			(* Case 60 - AspirazioneDX *)
			60: 
				IF AspirazioneSX1^.Status.CommandDone AND AspirazioneDX1^.Status.CommandDone AND
					AspirazioneSX2^.Status.CommandDone AND AspirazioneDX2^.Status.CommandDone THEN
					AspirazioneDX1^.Command^.Aspirazione_ON 	:= FALSE;
					AspirazioneDX1^.Command^.Aspirazione_OFF	:= FALSE;
					AspirazioneSX1^.Command^.Aspirazione_ON 	:= FALSE;
					AspirazioneSX1^.Command^.Aspirazione_OFF	:= FALSE;
					AspirazioneDX2^.Command^.Aspirazione_ON 	:= FALSE;
					AspirazioneDX2^.Command^.Aspirazione_OFF	:= FALSE;
					AspirazioneSX2^.Command^.Aspirazione_ON 	:= FALSE;
					AspirazioneSX2^.Command^.Aspirazione_OFF	:= FALSE;
					TFCommandCase(ADR(CmdExe),100,CommandCase_JMP);
				ELSIF AspirazioneSX1^.Status.ErrorID <> ErrNULL THEN
					TFClearAllCmdModulePinzaCompleta(AspirazioneDX1,AspirazioneSX1,AspirazioneDX2,AspirazioneSX2,CilindroApertura,CilindroSbloccoRotazione,CilindroSbloccoBascolante,AspirazioneFaldaDX,AspirazioneFaldaSX);
					TFError(ErrCYLINDER,AspirazioneSX1^.Status.ErrorID,ADR(CmdExe),ADR(State),ADR(Error),ADR(ErrorLog));
				ELSIF AspirazioneDX1^.Status.ErrorID <> ErrNULL THEN
					TFClearAllCmdModulePinzaCompleta(AspirazioneDX1,AspirazioneSX1,AspirazioneDX2,AspirazioneSX2,CilindroApertura,CilindroSbloccoRotazione,CilindroSbloccoBascolante,AspirazioneFaldaDX,AspirazioneFaldaSX);
					TFError(ErrCYLINDER,AspirazioneDX1^.Status.ErrorID,ADR(CmdExe),ADR(State),ADR(Error),ADR(ErrorLog));
				END_IF

			(* Case 70 - CilindroTasteggio *)
			70: 
				//IF CilindroTasteggio^.Status.CommandDone THEN
				//	CilindroTasteggio^.Command.Activation 		:= FALSE;
				//	CilindroTasteggio^.Command.Deactivation 	:= FALSE;
					TFCommandCase(ADR(CmdExe),100,CommandCase_JMP);
				//END_IF								
				
			(* Case 100 - End *)
			100:(* Clear All Output Here *)
				TFStateUpdate(ADR(State),StateMAN_END);
				TFCommandExeClear(ADR(CmdExe));

			ELSE
				TFError(ErrNOCMDCASE,ErrNULL,ADR(CmdExe),ADR(State),ADR(Error),ADR(ErrorLog));
		END_CASE;

		IF TFTimerDone(ADR(Timeout)) THEN
			TFClearAllCmdModulePinzaCompleta(AspirazioneDX1,AspirazioneSX1,AspirazioneDX2,AspirazioneSX2,CilindroApertura,CilindroSbloccoRotazione,CilindroSbloccoBascolante,AspirazioneFaldaDX,AspirazioneFaldaSX);
			TFError(ErrCMDTIMEOUT,ErrNULL,ADR(CmdExe),ADR(State),ADR(Error),ADR(ErrorLog));
		END_IF
	

	(* ******************************************************************************************************** *)
	(* PRELOAD - Presa del pezzo *)
	(* ******************************************************************************************************** *)
	CmdPRELOAD:
		CASE CmdExe.CmdCase OF
			
			(* Case 0 - Init Command*)
			0: 	TFStateUpdate(ADR(State),StatePRELOAD_RUN);
				TFTimerSet(ADR(Timeout),30000+200,TRUE);
				TFTimerSet(ADR(Timer),30000,TRUE);
				PrelievoSuCavallina := FALSE;
				StatoPinza.ElementoPrelevato := FALSE;
				IF TFCommandParRead(CmdExe.Cmd.Parameter,ADR(ParametersArray),2) THEN
					PrelievoSuCavallina	:= STRING_TO_BOOL(ParametersArray.Parameters[0]);
					AspiraSoloFalde		:= STRING_TO_BOOL(ParametersArray.Parameters[1]);
					TFCommandCase(ADR(CmdExe),10,CommandCase_JMP);
				ELSE
					TFError(ErrCMDPARNUM,ErrNULL,ADR(CmdExe),ADR(State),ADR(Error),ADR(ErrorLog));
					RETURN;
				END_IF;
				
			(* Case 10 - CilindroApertura *)
			10: 
				IF (ElementoInPrelievo.Typology = QUADROTTA OR ElementoInPrelievo.XDim >= 2700) AND AbilitaAperturaAutomaticaPinza THEN //sE HO LE CONDIZIONI APRO LA PINZA
					CilindroApertura^.Command.Activation 	:= TRUE;
					CilindroApertura^.Command.Deactivation 	:= FALSE;
	
					IF CilindroApertura^.Status.Active THEN
						CilindroApertura^.Command.Activation 	:= FALSE;
						CilindroApertura^.Command.Deactivation 	:= FALSE;
						TFCommandCase(ADR(CmdExe),20,CommandCase_JMP);
					ELSIF CilindroApertura^.Status.ErrorID <> ErrNULL THEN
						TFClearAllCmdModulePinzaCompleta(AspirazioneDX1,AspirazioneSX1,AspirazioneDX2,AspirazioneSX2,CilindroApertura,CilindroSbloccoRotazione,CilindroSbloccoBascolante,AspirazioneFaldaDX,AspirazioneFaldaSX);
						TFError(ErrCYLINDER,CilindroApertura^.Status.ErrorID,ADR(CmdExe),ADR(State),ADR(Error),ADR(ErrorLog));
					END_IF
				ELSE

					CilindroApertura^.Command.Activation 	:= FALSE;
					CilindroApertura^.Command.Deactivation 	:= TRUE;
	
					IF CilindroApertura^.Status.Inactive THEN
						CilindroApertura^.Command.Activation 	:= FALSE;
						CilindroApertura^.Command.Deactivation 	:= FALSE;
						TFCommandCase(ADR(CmdExe),20,CommandCase_JMP);
					ELSIF CilindroApertura^.Status.ErrorID <> ErrNULL THEN
						TFClearAllCmdModulePinzaCompleta(AspirazioneDX1,AspirazioneSX1,AspirazioneDX2,AspirazioneSX2,CilindroApertura,CilindroSbloccoRotazione,CilindroSbloccoBascolante,AspirazioneFaldaDX,AspirazioneFaldaSX);
						TFError(ErrCYLINDER,CilindroApertura^.Status.ErrorID,ADR(CmdExe),ADR(State),ADR(Error),ADR(ErrorLog));
					END_IF
					
				END_IF

			(* Case 20 - CilindroSbloccoRotazione *)
			20: 
				IF PrelievoSuCavallina THEN
					CilindroSbloccoRotazione^.Command.Activation 	:= AbilitazioneSbloccoRotazione;
					CilindroSbloccoRotazione^.Command.Deactivation 	:= FALSE;
	
					//CilindroTasteggio^.Command.Activation 		:= AbilitazioneCilindriTastatori;
					//CilindroTasteggio^.Command.Deactivation 	:= FALSE;
					
					IF (CilindroSbloccoRotazione^.Status.Active OR NOT AbilitazioneSbloccoRotazione) THEN
						CilindroSbloccoRotazione^.Command.Activation 	:= FALSE;
						CilindroSbloccoRotazione^.Command.Deactivation 	:= FALSE;
						//CilindroTasteggio^.Command.Activation 		:= FALSE;
						//CilindroTasteggio^.Command.Deactivation 	:= FALSE;
						TFCommandCase(ADR(CmdExe),30,CommandCase_JMP);
					ELSIF CilindroSbloccoRotazione^.Status.ErrorID <> ErrNULL AND AbilitazioneSbloccoRotazione THEN
						TFClearAllCmdModulePinzaCompleta(AspirazioneDX1,AspirazioneSX1,AspirazioneDX2,AspirazioneSX2,CilindroApertura,CilindroSbloccoRotazione,CilindroSbloccoBascolante,AspirazioneFaldaDX,AspirazioneFaldaSX);
						TFError(ErrCYLINDER,CilindroSbloccoRotazione^.Status.ErrorID,ADR(CmdExe),ADR(State),ADR(Error),ADR(ErrorLog));
					//ELSIF CilindroTasteggio^.Status.ErrorID <> ErrNULL THEN
					//	TFClearAllCmdModulePinzaCompleta(AspirazioneDX,AspirazioneSX,CilindroApertura,CilindroSbloccoRotazione,AspirazioneFaldaDX,AspirazioneFaldaSX);
					//	TFError(ErrCYLINDER,CilindroTasteggio^.Status.ErrorID,ADR(CmdExe),ADR(State),ADR(Error),ADR(ErrorLog));
					END_IF

				ELSE
					TFCommandCase(ADR(CmdExe),30,CommandCase_JMP);
				END_IF

			(* Case 30 - AspirazioneFaldaDX *)
			30: 

				IF NOT PrelievoSuCavallina AND AspiraSoloFalde THEN
					AspirazioneFaldaDX^.Command.Activation 	:= TRUE;
					AspirazioneFaldaDX^.Command.Deactivation 	:= FALSE;
					AspirazioneFaldaSX^.Command.Activation 	:= TRUE;
					AspirazioneFaldaSX^.Command.Deactivation 	:= FALSE;
					
					IF AspirazioneFaldaDX^.Status.Active AND AspirazioneFaldaSX^.Status.Active THEN
						AspirazioneFaldaDX^.Command.Activation 	:= FALSE;
						AspirazioneFaldaDX^.Command.Deactivation 	:= FALSE;
						AspirazioneFaldaSX^.Command.Activation 	:= FALSE;
						AspirazioneFaldaSX^.Command.Deactivation 	:= FALSE;
						TFCommandCase(ADR(CmdExe),40,CommandCase_JMP);
					ELSIF AspirazioneFaldaDX^.Status.ErrorID <> ErrNULL THEN
						TFClearAllCmdModulePinzaCompleta(AspirazioneDX1,AspirazioneSX1,AspirazioneDX2,AspirazioneSX2,CilindroApertura,CilindroSbloccoRotazione,CilindroSbloccoBascolante,AspirazioneFaldaDX,AspirazioneFaldaSX);
						TFError(ErrCYLINDER,AspirazioneFaldaDX^.Status.ErrorID,ADR(CmdExe),ADR(State),ADR(Error),ADR(ErrorLog));
					ELSIF AspirazioneFaldaSX^.Status.ErrorID <> ErrNULL THEN
						TFClearAllCmdModulePinzaCompleta(AspirazioneDX1,AspirazioneSX1,AspirazioneDX2,AspirazioneSX2,CilindroApertura,CilindroSbloccoRotazione,CilindroSbloccoBascolante,AspirazioneFaldaDX,AspirazioneFaldaSX);
						TFError(ErrCYLINDER,AspirazioneFaldaSX^.Status.ErrorID,ADR(CmdExe),ADR(State),ADR(Error),ADR(ErrorLog));
					END_IF
				ELSE
					TFCommandCase(ADR(CmdExe),40,CommandCase_JMP);
				END_IF


			(* Case 40 - AspirazioneDX + AspirazioneSX *)
			40: 
				AspirazioneDX1^.Command^.Aspirazione_ON 	:= TRUE;
				AspirazioneDX1^.Command^.Aspirazione_OFF := FALSE;
			
				AspirazioneSX1^.Command^.Aspirazione_ON 	:= TRUE;
				AspirazioneSX1^.Command^.Aspirazione_OFF := FALSE;
				
				AspirazioneDX2^.Command^.Aspirazione_ON 	:= TRUE;
				AspirazioneDX2^.Command^.Aspirazione_OFF := FALSE;
			
				AspirazioneSX2^.Command^.Aspirazione_ON 	:= TRUE;
				AspirazioneSX2^.Command^.Aspirazione_OFF := FALSE;
	
				IF AspirazioneDX1^.Status.CommandDone AND AspirazioneSX1^.Status.CommandDone AND
					AspirazioneDX2^.Status.CommandDone AND AspirazioneSX2^.Status.CommandDone THEN
						AspirazioneDX1^.Command^.Aspirazione_ON 	:= FALSE;
						AspirazioneDX1^.Command^.Aspirazione_OFF	:= FALSE;
						AspirazioneSX1^.Command^.Aspirazione_ON 	:= FALSE;
						AspirazioneSX1^.Command^.Aspirazione_OFF	:= FALSE;
						AspirazioneDX2^.Command^.Aspirazione_ON 	:= FALSE;
						AspirazioneDX2^.Command^.Aspirazione_OFF	:= FALSE;
						AspirazioneSX2^.Command^.Aspirazione_ON 	:= FALSE;
						AspirazioneSX2^.Command^.Aspirazione_OFF	:= FALSE;
					TFCommandCase(ADR(CmdExe),100,CommandCase_JMP);
				ELSIF AspirazioneSX1^.Status.ErrorID <> ErrNULL THEN
					TFClearAllCmdModulePinzaCompleta(AspirazioneDX1,AspirazioneSX1,AspirazioneDX2,AspirazioneSX2,CilindroApertura,CilindroSbloccoRotazione,CilindroSbloccoBascolante,AspirazioneFaldaDX,AspirazioneFaldaSX);
					TFError(ErrCYLINDER,AspirazioneSX1^.Status.ErrorID,ADR(CmdExe),ADR(State),ADR(Error),ADR(ErrorLog));
				ELSIF AspirazioneDX1^.Status.ErrorID <> ErrNULL THEN
					TFClearAllCmdModulePinzaCompleta(AspirazioneDX1,AspirazioneSX1,AspirazioneDX2,AspirazioneSX2,CilindroApertura,CilindroSbloccoRotazione,CilindroSbloccoBascolante,AspirazioneFaldaDX,AspirazioneFaldaSX);
					TFError(ErrCYLINDER,AspirazioneDX1^.Status.ErrorID,ADR(CmdExe),ADR(State),ADR(Error),ADR(ErrorLog));
				END_IF
				
			(* Case 100 *)
			100:TFStateUpdate(ADR(State),StatePRELOAD_END);
				TFCommandExeClear(ADR(CmdExe));

			ELSE
				TFError(ErrNOCMDCASE,ErrNULL,ADR(CmdExe),ADR(State),ADR(Error),ADR(ErrorLog));
		END_CASE

		IF TFTimerDone(ADR(Timeout)) THEN
			TFClearAllCmdModulePinzaCompleta(AspirazioneDX1,AspirazioneSX1,AspirazioneDX2,AspirazioneSX2,CilindroApertura,CilindroSbloccoRotazione,CilindroSbloccoBascolante,AspirazioneFaldaDX,AspirazioneFaldaSX);
			TFError(ErrCMDTIMEOUT,ErrNULL,ADR(CmdExe),ADR(State),ADR(Error),ADR(ErrorLog));
		END_IF
	


	(* ******************************************************************************************************** *)
	(* CHECKPRESENCE -  *)
	(* ******************************************************************************************************** *)
	CmdCHECKPRESENCE:
		CASE CmdExe.CmdCase OF
			
			(* Case 0 - Init Command*)
			0: 	TFStateUpdate(ADR(State),StateCHECKPRESENCE_RUN);
				TFTimerSet(ADR(Timeout),60000.0+100+HMI_TempoControlloPresaPiastrella,TRUE);
				TFTimerSet(ADR(Timer),2000.0+HMI_TempoControlloPresaPiastrella,TRUE);
				TFTimerSet(ADR(TimerPresaPiastrella),HMI_TempoControlloPresaPiastrella,TRUE);
				StatoPinza.ElementoPrelevato := FALSE;
				CilindroSbloccoRotazione^.Command.Activation 	:= FALSE;
				CilindroSbloccoRotazione^.Command.Deactivation 	:= TRUE;

				TFCommandCase(ADR(CmdExe),1,CommandCase_INC);
				
			(* Case 1 - *)					
			1:
				StatoPinza.ElementoPrelevato := FALSE;
				IF CilindroSbloccoRotazione^.Status.Inactive THEN
					CilindroSbloccoRotazione^.Command.Activation 	:= FALSE;
					CilindroSbloccoRotazione^.Command.Deactivation 	:= TRUE;	
				END_IF

			IF IN.ByPassSensoreVuoto OR TFTimerDone(ADR(TimerPresaPiastrella)) THEN 
					//Tutte piastrelle o tutte falde
					IF ((AspirazioneDX1^.Status.DepressioneSoglia1_OK AND AspirazioneSX1^.Status.DepressioneSoglia1_OK) AND
						(AspirazioneDX2^.Status.DepressioneSoglia1_OK AND AspirazioneSX2^.Status.DepressioneSoglia1_OK)) OR
						((AspirazioneFaldaDX^.Status.Active AND IN.TastoreCartoneDX AND FTC_FaldaDXFiltrata) AND
						(AspirazioneFaldaSX^.Status.Active AND IN.TastoreCartoneSX AND FTC_FaldaSXFiltrata)) OR
						IN.ByPassSensoreVuoto THEN
							StatoPinza.ElementoPrelevato := TRUE;
							TFCommandCase(ADR(CmdExe),1,CommandCase_INC);
					ELSIF TFTimerDone(ADR(TimerPresaPiastrella)) THEN
						TFCommandCase(ADR(CmdExe),1,CommandCase_INC);
						StatoPinza.ElementoPrelevato := FALSE;	
					END_IF			
				ELSIF TFTimerDone(ADR(TimerPresaPiastrella)) THEN
					TFCommandCase(ADR(CmdExe),1,CommandCase_INC);
					StatoPinza.ElementoPrelevato := FALSE;
				END_IF			
				IF TFTimerDone(ADR(Timer)) THEN
					TFClearAllCmdModulePinzaCompleta(AspirazioneDX1,AspirazioneSX1,AspirazioneDX2,AspirazioneSX2,CilindroApertura,CilindroSbloccoRotazione,CilindroSbloccoBascolante,AspirazioneFaldaDX,AspirazioneFaldaSX);
					TFError(ErrMalfunzionamentoSensoriPresenzaPinza,ErrNULL,ADR(CmdExe),ADR(State),ADR(Error),ADR(ErrorLog));
				ELSIF TFTimerDone(ADR(Timeout)) THEN
					TFClearAllCmdModulePinzaCompleta(AspirazioneDX1,AspirazioneSX1,AspirazioneDX2,AspirazioneSX2,CilindroApertura,CilindroSbloccoRotazione,CilindroSbloccoBascolante,AspirazioneFaldaDX,AspirazioneFaldaSX);
					TFError(ErrCMDTIMEOUT,ErrNULL,ADR(CmdExe),ADR(State),ADR(Error),ADR(ErrorLog));
				END_IF
		
			(* Case 2 - *)		
			2: 
				TFTimerSet(ADR(TimerAspirazione),1,TRUE);
				TFCommandCase(ADR(CmdExe),1,CommandCase_INC);
				IF TFTimerDone(ADR(Timer)) THEN
					TFClearAllCmdModulePinzaCompleta(AspirazioneDX1,AspirazioneSX1,AspirazioneDX2,AspirazioneSX2,CilindroApertura,CilindroSbloccoRotazione,CilindroSbloccoBascolante,AspirazioneFaldaDX,AspirazioneFaldaSX);
					TFError(ErrMalfunzionamentoSensoriPresenzaPinza,ErrNULL,ADR(CmdExe),ADR(State),ADR(Error),ADR(ErrorLog));
				ELSIF TFTimerDone(ADR(Timeout)) THEN
					TFClearAllCmdModulePinzaCompleta(AspirazioneDX1,AspirazioneSX1,AspirazioneDX2,AspirazioneSX2,CilindroApertura,CilindroSbloccoRotazione,CilindroSbloccoBascolante,AspirazioneFaldaDX,AspirazioneFaldaSX);
					TFError(ErrCMDTIMEOUT,ErrNULL,ADR(CmdExe),ADR(State),ADR(Error),ADR(ErrorLog));
				END_IF				
				
			3:
				IF TFTimerDone(ADR(TimerAspirazione)) THEN
					TFStateUpdate(ADR(State),StateCHECKPRESENCE_RUN+10);
					TFCommandCase(ADR(CmdExe),100,CommandCase_JMP);
				END_IF
				
			4:			
				IF 	((AspirazioneFaldaDX^.Status.Active AND IN.TastoreCartoneDX AND FTC_FaldaDXFiltrata AND NOT AspirazioneDX1^.Status.DepressioneSoglia1_OK) OR
					(AspirazioneFaldaSX^.Status.Active AND IN.TastoreCartoneSX AND FTC_FaldaSXFiltrata AND NOT AspirazioneSX1^.Status.DepressioneSoglia1_OK)) THEN
					StatoPinza.ElementoPrelevato := TRUE;
					TFCommandCase(ADR(CmdExe),100,CommandCase_JMP);
				ELSE
					TFCommandCase(ADR(CmdExe),100,CommandCase_JMP);
					StatoPinza.ElementoPrelevato := FALSE;
				END_IF	
			
			(* Case 100 *)
			100:TFStateUpdate(ADR(State),StateCHECKPRESENCE_END);
				TFCommandExeClear(ADR(CmdExe));

			ELSE
				TFError(ErrNOCMDCASE,ErrNULL,ADR(CmdExe),ADR(State),ADR(Error),ADR(ErrorLog));
		END_CASE

	(* ******************************************************************************************************** *)
	(* CmdSbloccaBascolante - SGANCIO BASCULANTE *)
	(* ******************************************************************************************************** *)
	CmdSbloccaBascolante:
		CASE CmdExe.CmdCase OF
			
			(* Case 0 - Init Command*)
			0: 	TFStateUpdate(ADR(State),StateSbloccaBascolante_RUN);
				TFTimerSet(ADR(Timeout),30000+200,TRUE);
				TFTimerSet(ADR(Timer),30000,TRUE);
				//IF NOT IN_SimulazioneSenzaHW THEN
					TFCommandCase(ADR(CmdExe),10,CommandCase_JMP);
				//ELSE
				//	TFCommandCase(ADR(CmdExe),100,CommandCase_JMP);
				//END_IF
				
			(* Case 10 - CilindroSblocco bacolante *)
			10: 
				CilindroSbloccoBascolante^.Command.Activation 	:= AbilitazioneSbloccoBascolante;
				CilindroSbloccoBascolante^.Command.Deactivation := FALSE;

				IF (CilindroSbloccoBascolante^.Status.Active OR NOT AbilitazioneSbloccoBascolante)THEN
					CilindroSbloccoBascolante^.Command.Activation 	:= FALSE;
					CilindroSbloccoBascolante^.Command.Deactivation 	:= FALSE;
					TFCommandCase(ADR(CmdExe),100,CommandCase_JMP);
				ELSIF CilindroSbloccoBascolante^.Status.ErrorID <> ErrNULL AND AbilitazioneSbloccoBascolante THEN
					TFClearAllCmdModulePinzaCompleta(AspirazioneDX1,AspirazioneSX1,AspirazioneDX2,AspirazioneSX2,CilindroApertura,CilindroSbloccoRotazione,CilindroSbloccoBascolante,AspirazioneFaldaDX,AspirazioneFaldaSX);
					TFError(ErrCYLINDER,CilindroSbloccoBascolante^.Status.ErrorID,ADR(CmdExe),ADR(State),ADR(Error),ADR(ErrorLog));
				END_IF

				
			(* Case 100 *)
			100:TFStateUpdate(ADR(State),StateSbloccaBascolante_END);
				TFCommandExeClear(ADR(CmdExe));

			ELSE
				TFError(ErrNOCMDCASE,ErrNULL,ADR(CmdExe),ADR(State),ADR(Error),ADR(ErrorLog));
		END_CASE

		IF TFTimerDone(ADR(Timeout)) THEN
			TFClearAllCmdModulePinzaCompleta(AspirazioneDX1,AspirazioneSX1,AspirazioneDX2,AspirazioneSX2,CilindroApertura,CilindroSbloccoRotazione,CilindroSbloccoBascolante,AspirazioneFaldaDX,AspirazioneFaldaSX);
			TFError(ErrCMDTIMEOUT,ErrNULL,ADR(CmdExe),ADR(State),ADR(Error),ADR(ErrorLog));
		END_IF
		
		(* ******************************************************************************************************** *)
	(* CmdBloccaBascolante - AGGANCIO BASCULANTE *)
	(* ******************************************************************************************************** *)
	CmdBloccaBascolante:
		CASE CmdExe.CmdCase OF
			
			(* Case 0 - Init Command*)
			0: 	TFStateUpdate(ADR(State),StateBloccaBascolante_RUN);
				TFTimerSet(ADR(Timeout),30000+200,TRUE);
				TFTimerSet(ADR(Timer),30000,TRUE);
				//IF NOT IN_SimulazioneSenzaHW THEN
					TFCommandCase(ADR(CmdExe),10,CommandCase_JMP);
				//ELSE
				//	TFCommandCase(ADR(CmdExe),100,CommandCase_JMP);
				//END_IF
				
			(* Case 10 - CilindroSblocco bacolante *)
			10: 
				CilindroSbloccoBascolante^.Command.Activation 	:= FALSE;
				CilindroSbloccoBascolante^.Command.Deactivation := TRUE;

				IF  CilindroSbloccoBascolante^.Status.Inactive THEN
					CilindroSbloccoBascolante^.Command.Activation 	:= FALSE;
					CilindroSbloccoBascolante^.Command.Deactivation := FALSE;
					TFCommandCase(ADR(CmdExe),100,CommandCase_JMP);
				ELSIF CilindroSbloccoBascolante^.Status.ErrorID <> ErrNULL AND AbilitazioneSbloccoBascolante THEN
					TFClearAllCmdModulePinzaCompleta(AspirazioneDX1,AspirazioneSX1,AspirazioneDX2,AspirazioneSX2,CilindroApertura,CilindroSbloccoRotazione,CilindroSbloccoBascolante,AspirazioneFaldaDX,AspirazioneFaldaSX);
					TFError(ErrCYLINDER,CilindroSbloccoBascolante^.Status.ErrorID,ADR(CmdExe),ADR(State),ADR(Error),ADR(ErrorLog));
				END_IF

				
			(* Case 100 *)
			100:TFStateUpdate(ADR(State),StateBloccaBascolante_END);
				TFCommandExeClear(ADR(CmdExe));

			ELSE
				TFError(ErrNOCMDCASE,ErrNULL,ADR(CmdExe),ADR(State),ADR(Error),ADR(ErrorLog));
		END_CASE

		IF TFTimerDone(ADR(Timeout)) THEN
			TFClearAllCmdModulePinzaCompleta(AspirazioneDX1,AspirazioneSX1,AspirazioneDX2,AspirazioneSX2,CilindroApertura,CilindroSbloccoRotazione,CilindroSbloccoBascolante,AspirazioneFaldaDX,AspirazioneFaldaSX);
			TFError(ErrCMDTIMEOUT,ErrNULL,ADR(CmdExe),ADR(State),ADR(Error),ADR(ErrorLog));
		END_IF
		
	(* ******************************************************************************************************** *)
	(* CmdSbloccaRotazione - SGANCIO rotazione *)
	(* ******************************************************************************************************** *)
	CmdSbloccaRotazione:
		CASE CmdExe.CmdCase OF
			
			(* Case 0 - Init Command*)
			0: 	TFStateUpdate(ADR(State),StateSbloccaRotazione_RUN);
				TFTimerSet(ADR(Timeout),30000+200,TRUE);
				TFTimerSet(ADR(Timer),30000,TRUE);
				//IF NOT IN_SimulazioneSenzaHW THEN
					TFCommandCase(ADR(CmdExe),10,CommandCase_JMP);
				//ELSE
				//	TFCommandCase(ADR(CmdExe),100,CommandCase_JMP);
				//END_IF
				
			(* Case 10 - CilindroSblocco bacolante *)
			10: 
				CilindroSbloccoRotazione^.Command.Activation 	:= AbilitazioneSbloccoRotazione;
				CilindroSbloccoRotazione^.Command.Deactivation := FALSE;

				IF (CilindroSbloccoRotazione^.Status.Active OR NOT AbilitazioneSbloccoRotazione)THEN
					CilindroSbloccoRotazione^.Command.Activation 	:= FALSE;
					CilindroSbloccoRotazione^.Command.Deactivation 	:= FALSE;
					TFCommandCase(ADR(CmdExe),100,CommandCase_JMP);
				ELSIF CilindroSbloccoBascolante^.Status.ErrorID <> ErrNULL AND AbilitazioneSbloccoRotazione THEN
					TFClearAllCmdModulePinzaCompleta(AspirazioneDX1,AspirazioneSX1,AspirazioneDX2,AspirazioneSX2,CilindroApertura,CilindroSbloccoRotazione,CilindroSbloccoBascolante,AspirazioneFaldaDX,AspirazioneFaldaSX);
					TFError(ErrCYLINDER,CilindroSbloccoRotazione^.Status.ErrorID,ADR(CmdExe),ADR(State),ADR(Error),ADR(ErrorLog));
				END_IF

				
			(* Case 100 *)
			100:TFStateUpdate(ADR(State),StateSbloccaRotazione_END);
				TFCommandExeClear(ADR(CmdExe));

			ELSE
				TFError(ErrNOCMDCASE,ErrNULL,ADR(CmdExe),ADR(State),ADR(Error),ADR(ErrorLog));
		END_CASE

		IF TFTimerDone(ADR(Timeout)) THEN
			TFClearAllCmdModulePinzaCompleta(AspirazioneDX1,AspirazioneSX1,AspirazioneDX2,AspirazioneSX2,CilindroApertura,CilindroSbloccoRotazione,CilindroSbloccoBascolante,AspirazioneFaldaDX,AspirazioneFaldaSX);
			TFError(ErrCMDTIMEOUT,ErrNULL,ADR(CmdExe),ADR(State),ADR(Error),ADR(ErrorLog));
		END_IF
		
	(* ******************************************************************************************************** *)
	(* CmdBloccaROTAZIONE - BLOCCA ROTAZIONE *)
	(* ******************************************************************************************************** *)
	CmdBloccaRotazione:
		CASE CmdExe.CmdCase OF
			
			(* Case 0 - Init Command*)
			0: 	TFStateUpdate(ADR(State),StateBloccaRotazione_RUN);
				TFTimerSet(ADR(Timeout),30000+200,TRUE);
				TFTimerSet(ADR(Timer),30000,TRUE);
				//IF NOT IN_SimulazioneSenzaHW THEN
					TFCommandCase(ADR(CmdExe),10,CommandCase_JMP);
				//ELSE
				//	TFCommandCase(ADR(CmdExe),100,CommandCase_JMP);
				//END_IF
				
			(* Case 10 - CilindroSblocco bacolante *)
			10: 
				CilindroSbloccoRotazione^.Command.Activation 	:= FALSE;
				CilindroSbloccoRotazione^.Command.Deactivation  := TRUE;

				IF (CilindroSbloccoRotazione^.Status.Inactive) THEN
					CilindroSbloccoRotazione^.Command.Activation 	:= FALSE;
					CilindroSbloccoRotazione^.Command.Deactivation := FALSE;
					TFCommandCase(ADR(CmdExe),100,CommandCase_JMP);
				ELSIF CilindroSbloccoBascolante^.Status.ErrorID <> ErrNULL THEN
					TFClearAllCmdModulePinzaCompleta(AspirazioneDX1,AspirazioneSX1,AspirazioneDX2,AspirazioneSX2,CilindroApertura,CilindroSbloccoRotazione,CilindroSbloccoBascolante,AspirazioneFaldaDX,AspirazioneFaldaSX);
					TFError(ErrCYLINDER,CilindroSbloccoBascolante^.Status.ErrorID,ADR(CmdExe),ADR(State),ADR(Error),ADR(ErrorLog));
				END_IF

				
			(* Case 100 *)
			100:TFStateUpdate(ADR(State),StateBloccaBascolante_END);
				TFCommandExeClear(ADR(CmdExe));

			ELSE
				TFError(ErrNOCMDCASE,ErrNULL,ADR(CmdExe),ADR(State),ADR(Error),ADR(ErrorLog));
		END_CASE

		IF TFTimerDone(ADR(Timeout)) THEN
			TFClearAllCmdModulePinzaCompleta(AspirazioneDX1,AspirazioneSX1,AspirazioneDX2,AspirazioneSX2,CilindroApertura,CilindroSbloccoRotazione,CilindroSbloccoBascolante,AspirazioneFaldaDX,AspirazioneFaldaSX);
			TFError(ErrCMDTIMEOUT,ErrNULL,ADR(CmdExe),ADR(State),ADR(Error),ADR(ErrorLog));
		END_IF
		
	(* ******************************************************************************************************** *)
	(* CmdBloccaPinza- BLOCCA ROTAZIONE + BLOCCA BASCULANTE *)
	(* ******************************************************************************************************** *)
	CmdBloccaPinza:
		CASE CmdExe.CmdCase OF
			
			(* Case 0 - Init Command*)
			0: 	TFStateUpdate(ADR(State),StateBloccaPinza_RUN);
				TFTimerSet(ADR(Timeout),30000+200,TRUE);
				TFTimerSet(ADR(Timer),30000,TRUE);
				//IF NOT IN_SimulazioneSenzaHW THEN
					TFCommandCase(ADR(CmdExe),10,CommandCase_JMP);
				//ELSE
				//	TFCommandCase(ADR(CmdExe),100,CommandCase_JMP);
				//END_IF
				
			(* Case 10 - CilindroSblocco bascolante + rotazione *)
			10: 
				CilindroSbloccoRotazione^.Command.Activation 	:= FALSE;
				CilindroSbloccoRotazione^.Command.Deactivation  := TRUE;
				
				CilindroSbloccoBascolante^.Command.Activation 	:= FALSE;
				CilindroSbloccoBascolante^.Command.Deactivation  := TRUE;

				IF (CilindroSbloccoRotazione^.Status.Inactive) AND CilindroSbloccoRotazione^.Status.Inactive THEN
					CilindroSbloccoRotazione^.Command.Activation 	:= FALSE;
					CilindroSbloccoRotazione^.Command.Deactivation := FALSE;
					CilindroSbloccoBascolante^.Command.Activation 	:= FALSE;
					CilindroSbloccoBascolante^.Command.Deactivation  := FALSE;

					TFCommandCase(ADR(CmdExe),100,CommandCase_JMP);
				ELSIF CilindroSbloccoBascolante^.Status.ErrorID <> ErrNULL THEN
					TFClearAllCmdModulePinzaCompleta(AspirazioneDX1,AspirazioneSX1,AspirazioneDX2,AspirazioneSX2,CilindroApertura,CilindroSbloccoRotazione,CilindroSbloccoBascolante,AspirazioneFaldaDX,AspirazioneFaldaSX);
					TFError(ErrCYLINDER,CilindroSbloccoBascolante^.Status.ErrorID,ADR(CmdExe),ADR(State),ADR(Error),ADR(ErrorLog));
				ELSIF CilindroSbloccoRotazione^.Status.ErrorID <> ErrNULL THEN
					TFClearAllCmdModulePinzaCompleta(AspirazioneDX1,AspirazioneSX1,AspirazioneDX2,AspirazioneSX2,CilindroApertura,CilindroSbloccoRotazione,CilindroSbloccoBascolante,AspirazioneFaldaDX,AspirazioneFaldaSX);
					TFError(ErrCYLINDER,CilindroSbloccoRotazione^.Status.ErrorID,ADR(CmdExe),ADR(State),ADR(Error),ADR(ErrorLog));
				END_IF

				
			(* Case 100 *)
			100:TFStateUpdate(ADR(State),StateBloccaPinza_END);
				TFCommandExeClear(ADR(CmdExe));

			ELSE
				TFError(ErrNOCMDCASE,ErrNULL,ADR(CmdExe),ADR(State),ADR(Error),ADR(ErrorLog));
		END_CASE

		IF TFTimerDone(ADR(Timeout)) THEN
			TFClearAllCmdModulePinzaCompleta(AspirazioneDX1,AspirazioneSX1,AspirazioneDX2,AspirazioneSX2,CilindroApertura,CilindroSbloccoRotazione,CilindroSbloccoBascolante,AspirazioneFaldaDX,AspirazioneFaldaSX);
			TFError(ErrCMDTIMEOUT,ErrNULL,ADR(CmdExe),ADR(State),ADR(Error),ADR(ErrorLog));
		END_IF

	
	(* ******************************************************************************************************** *)
	(* CmdSbloccaPinza- SBLOCCA ROTAZIONE + SBLOCCA BASCULANTE *)
	(* ******************************************************************************************************** *)
	CmdSbloccaPinza:
			CASE CmdExe.CmdCase OF
				
				(* Case 0 - Init Command*)
				0: 	TFStateUpdate(ADR(State),StateSbloccaPinza_RUN);
					TFTimerSet(ADR(Timeout),30000+200,TRUE);
					TFTimerSet(ADR(Timer),30000,TRUE);
					//IF NOT IN_SimulazioneSenzaHW THEN
						TFCommandCase(ADR(CmdExe),10,CommandCase_JMP);
					//ELSE
					//	TFCommandCase(ADR(CmdExe),100,CommandCase_JMP);
					//END_IF
					
				(* Case 10 - CilindroSblocco bascolante + rotazione *)
				10: 
					CilindroSbloccoBascolante^.Command.Activation 	:= AbilitazioneSbloccoBascolante;
					CilindroSbloccoBascolante^.Command.Deactivation := FALSE;
					CilindroSbloccoRotazione^.Command.Activation 	:= AbilitazioneSbloccoRotazione;
					CilindroSbloccoRotazione^.Command.Deactivation  := FALSE;
	
					IF (CilindroSbloccoBascolante^.Status.Active OR NOT AbilitazioneSbloccoBascolante) AND 
						(CilindroSbloccoRotazione^.Status.Active OR NOT AbilitazioneSbloccoRotazione) THEN
							CilindroSbloccoBascolante^.Command.Activation 	:= FALSE;
							CilindroSbloccoBascolante^.Command.Deactivation := FALSE;
							CilindroSbloccoRotazione^.Command.Activation 	:= FALSE;
							CilindroSbloccoRotazione^.Command.Deactivation  := FALSE;
							TFCommandCase(ADR(CmdExe),100,CommandCase_JMP);
					ELSIF CilindroSbloccoBascolante^.Status.ErrorID <> ErrNULL AND AbilitazioneSbloccoBascolante THEN
						TFClearAllCmdModulePinzaCompleta(AspirazioneDX1,AspirazioneSX1,AspirazioneDX2,AspirazioneSX2,CilindroApertura,CilindroSbloccoRotazione,CilindroSbloccoBascolante,AspirazioneFaldaDX,AspirazioneFaldaSX);
						TFError(ErrCYLINDER,CilindroSbloccoBascolante^.Status.ErrorID,ADR(CmdExe),ADR(State),ADR(Error),ADR(ErrorLog));
					ELSIF CilindroSbloccoRotazione^.Status.ErrorID <> ErrNULL THEN
						TFClearAllCmdModulePinzaCompleta(AspirazioneDX1,AspirazioneSX1,AspirazioneDX2,AspirazioneSX2,CilindroApertura,CilindroSbloccoRotazione,CilindroSbloccoBascolante,AspirazioneFaldaDX,AspirazioneFaldaSX);
						TFError(ErrCYLINDER,CilindroSbloccoRotazione^.Status.ErrorID,ADR(CmdExe),ADR(State),ADR(Error),ADR(ErrorLog));
					END_IF
					
				(* Case 100 *)
				100:TFStateUpdate(ADR(State),StateSbloccaPinza_END);
					TFCommandExeClear(ADR(CmdExe));
	
				ELSE
					TFError(ErrNOCMDCASE,ErrNULL,ADR(CmdExe),ADR(State),ADR(Error),ADR(ErrorLog));
			END_CASE
	
			IF TFTimerDone(ADR(Timeout)) THEN
				TFClearAllCmdModulePinzaCompleta(AspirazioneDX1,AspirazioneSX1,AspirazioneDX2,AspirazioneSX2,CilindroApertura,CilindroSbloccoRotazione,CilindroSbloccoBascolante,AspirazioneFaldaDX,AspirazioneFaldaSX);
				TFError(ErrCMDTIMEOUT,ErrNULL,ADR(CmdExe),ADR(State),ADR(Error),ADR(ErrorLog));
			END_IF
	
	(* ******************************************************************************************************** *)
	(* UNLOAD - Disattivazione aspirazione *)
	(* ******************************************************************************************************** *)
	CmdUNLOAD:
		CASE CmdExe.CmdCase OF
			
			(* Case 0 - Init Command*)
			0: 	TFStateUpdate(ADR(State),StateUNLOAD_RUN);
				TFTimerSet(ADR(Timeout),30000+200,TRUE);
				TFTimerSet(ADR(Timer),30000,TRUE);
				DisattivazioneTotaleAspirazioni := FALSE;
				
				IF Mission^.State = MISSION_STATE_DEPOSITO_FALDA_DEPAL_RUN THEN
					TFCommandCase(ADR(CmdExe),10,CommandCase_JMP);
				ELSIF Mission^.State = MISSION_STATE_DEPOSITO_LASTRA_DEPAL_RUN THEN
		
					IF NOT StatoPinza.LatoDxFaldaInPresa AND NOT StatoPinza.LatoSxFaldaInPresa THEN
						StatoPinza.ElementoPrelevato := FALSE;
						DisattivazioneTotaleAspirazioni := TRUE;
						TFCommandCase(ADR(CmdExe),10,CommandCase_JMP);
					ELSE
						TFCommandCase(ADR(CmdExe),20,CommandCase_JMP);
					END_IF					
				ELSE
					DisattivazioneTotaleAspirazioni := TRUE;
					StatoPinza.ElementoPrelevato := FALSE;
					TFCommandCase(ADR(CmdExe),10,CommandCase_JMP);
				END_IF
				
			(* Case 10 - Disattivazione Aspirazione falde *)					
			10:	
				AspirazioneFaldaDX^.Command.Activation 		:= FALSE;
				AspirazioneFaldaDX^.Command.Deactivation 	:= TRUE;
				AspirazioneFaldaSX^.Command.Activation 		:= FALSE;
				AspirazioneFaldaSX^.Command.Deactivation 	:= TRUE;

				CilindroSbloccoRotazione^.Command.Activation 	:= FALSE;
				CilindroSbloccoRotazione^.Command.Deactivation 	:= TRUE;
				
				IF AspirazioneFaldaDX^.Status.Inactive AND AspirazioneFaldaSX^.Status.Inactive AND CilindroSbloccoRotazione^.Status.Inactive THEN
					AspirazioneFaldaDX^.Command.Activation 		:= FALSE;
					AspirazioneFaldaDX^.Command.Deactivation 	:= FALSE;
					AspirazioneFaldaSX^.Command.Activation 		:= FALSE;
					AspirazioneFaldaSX^.Command.Deactivation 	:= FALSE;
					CilindroSbloccoRotazione^.Command.Activation 	:= FALSE;
					CilindroSbloccoRotazione^.Command.Deactivation 	:= FALSE;
					IF DisattivazioneTotaleAspirazioni THEN
						TFCommandCase(ADR(CmdExe),20,CommandCase_JMP);
					ELSE
						TFCommandCase(ADR(CmdExe),100,CommandCase_JMP);
					END_IF				
				ELSIF AspirazioneFaldaDX^.Status.ErrorID <> ErrNULL THEN
					TFClearAllCmdModulePinzaCompleta(AspirazioneDX1,AspirazioneSX1,AspirazioneDX2,AspirazioneSX2,CilindroApertura,CilindroSbloccoRotazione,CilindroSbloccoBascolante,AspirazioneFaldaDX,AspirazioneFaldaSX);					TFError(ErrCYLINDER,AspirazioneFaldaDX^.Status.ErrorID,ADR(CmdExe),ADR(State),ADR(Error),ADR(ErrorLog));
				ELSIF AspirazioneFaldaSX^.Status.ErrorID <> ErrNULL THEN
					TFClearAllCmdModulePinzaCompleta(AspirazioneDX1,AspirazioneSX1,AspirazioneDX2,AspirazioneSX2,CilindroApertura,CilindroSbloccoRotazione,CilindroSbloccoBascolante,AspirazioneFaldaDX,AspirazioneFaldaSX);					TFError(ErrCYLINDER,AspirazioneFaldaSX^.Status.ErrorID,ADR(CmdExe),ADR(State),ADR(Error),ADR(ErrorLog));
				ELSIF CilindroSbloccoRotazione^.Status.ErrorID <> ErrNULL THEN
					TFClearAllCmdModulePinzaCompleta(AspirazioneDX1,AspirazioneSX1,AspirazioneDX2,AspirazioneSX2,CilindroApertura,CilindroSbloccoRotazione,CilindroSbloccoBascolante,AspirazioneFaldaDX,AspirazioneFaldaSX);					TFError(ErrCYLINDER,CilindroSbloccoRotazione^.Status.ErrorID,ADR(CmdExe),ADR(State),ADR(Error),ADR(ErrorLog));
				END_IF
			
			(* Case 20 - Disattivazione aspirazione piastrella *)		
			20: 
				AspirazioneDX1^.Command^.Aspirazione_ON 	:= FALSE;
				AspirazioneDX1^.Command^.Aspirazione_OFF := TRUE;
				AspirazioneSX1^.Command^.Aspirazione_ON 	:= FALSE;
				AspirazioneSX1^.Command^.Aspirazione_OFF := TRUE;
				
				AspirazioneDX2^.Command^.Aspirazione_ON  := FALSE;
				AspirazioneDX2^.Command^.Aspirazione_OFF := TRUE;
				AspirazioneSX2^.Command^.Aspirazione_ON  := FALSE;
				AspirazioneSX2^.Command^.Aspirazione_OFF := TRUE;
		
				IF AspirazioneDX1^.Status.CommandDone AND AspirazioneSX1^.Status.CommandDone AND
					AspirazioneDX2^.Status.CommandDone AND AspirazioneSX2^.Status.CommandDone THEN
						AspirazioneDX1^.Command^.Aspirazione_ON 	:= FALSE;
						AspirazioneDX1^.Command^.Aspirazione_OFF	:= FALSE;
						AspirazioneSX1^.Command^.Aspirazione_ON 	:= FALSE;
						AspirazioneSX1^.Command^.Aspirazione_OFF	:= FALSE;
						AspirazioneDX2^.Command^.Aspirazione_ON 	:= FALSE;
						AspirazioneDX2^.Command^.Aspirazione_OFF	:= FALSE;
						AspirazioneSX2^.Command^.Aspirazione_ON 	:= FALSE;
						AspirazioneSX2^.Command^.Aspirazione_OFF	:= FALSE;
					TFTimerSet(ADR(TimerAspirazione),HMI_TempoRilascioInDeposito,TRUE);
					TFCommandCase(ADR(CmdExe),30,CommandCase_JMP);
				ELSIF AspirazioneSX1^.Status.ErrorID <> ErrNULL THEN
					TFClearAllCmdModulePinzaCompleta(AspirazioneDX1,AspirazioneSX1,AspirazioneDX2,AspirazioneSX2,CilindroApertura,CilindroSbloccoRotazione,CilindroSbloccoBascolante,AspirazioneFaldaDX,AspirazioneFaldaSX);
					TFError(ErrCYLINDER,AspirazioneSX1^.Status.ErrorID,ADR(CmdExe),ADR(State),ADR(Error),ADR(ErrorLog));
				ELSIF AspirazioneDX1^.Status.ErrorID <> ErrNULL THEN
					TFClearAllCmdModulePinzaCompleta(AspirazioneDX1,AspirazioneSX1,AspirazioneDX2,AspirazioneSX2,CilindroApertura,CilindroSbloccoRotazione,CilindroSbloccoBascolante,AspirazioneFaldaDX,AspirazioneFaldaSX);					TFError(ErrCYLINDER,AspirazioneDX1^.Status.ErrorID,ADR(CmdExe),ADR(State),ADR(Error),ADR(ErrorLog));
				END_IF
			
			(* Case 30 - Attesa tempo distacco *)		
			30:
				IF TFTimerDone(ADR(TimerAspirazione)) THEN
					IF IN.RichiestaRicalibrazioneOvemEsterna AND NOT IN.ByPassSensoreVuoto THEN
						IN.RichiestaRicalibrazioneOvemEsterna := FALSE;
						TFCommandCase(ADR(CmdExe),40,CommandCase_JMP);
					ELSE
						TFCommandCase(ADR(CmdExe),100,CommandCase_JMP);
					END_IF		
				END_IF
				
			(* Case 40 - Attesa tempo distacco *)		
			40:	
				AspirazioneDX1^.Command^.Aspirazione_ON_ScritturaSoglia 	:= TRUE;
				AspirazioneSX1^.Command^.Aspirazione_ON_ScritturaSoglia 	:= TRUE;
				AspirazioneDX2^.Command^.Aspirazione_ON_ScritturaSoglia 	:= TRUE;
				AspirazioneSX2^.Command^.Aspirazione_ON_ScritturaSoglia 	:= TRUE;
				IF AspirazioneDX1^.Status.CommandDone AND AspirazioneSX1^.Status.CommandDone AND
					AspirazioneDX2^.Status.CommandDone AND AspirazioneSX2^.Status.CommandDone THEN
						AspirazioneDX1^.Command^.Aspirazione_ON_ScritturaSoglia		:= FALSE;
						AspirazioneSX1^.Command^.Aspirazione_ON_ScritturaSoglia		:= FALSE;
						AspirazioneDX2^.Command^.Aspirazione_ON_ScritturaSoglia		:= FALSE;
						AspirazioneSX2^.Command^.Aspirazione_ON_ScritturaSoglia		:= FALSE;
						TFCommandCase(ADR(CmdExe),100,CommandCase_JMP);
				ELSIF TFTimerDone(ADR(Timer)) THEN
					AspirazioneDX1^.Command^.Aspirazione_ON_ScritturaSoglia		:= FALSE;
					AspirazioneSX1^.Command^.Aspirazione_ON_ScritturaSoglia		:= FALSE;
					AspirazioneDX2^.Command^.Aspirazione_ON_ScritturaSoglia		:= FALSE;
					AspirazioneSX2^.Command^.Aspirazione_ON_ScritturaSoglia		:= FALSE;
					TFError(ErrTOHOME,ErrNULL,ADR(CmdExe),ADR(State),ADR(Error),ADR(ErrorLog));
				END_IF
				
		
			(* Case 100 *)
			100:TFStateUpdate(ADR(State),StateUNLOAD_END);
				TFCommandExeClear(ADR(CmdExe));

			ELSE
				TFError(ErrNOCMDCASE,ErrNULL,ADR(CmdExe),ADR(State),ADR(Error),ADR(ErrorLog));
		END_CASE

		IF TFTimerDone(ADR(Timeout)) THEN
			TFClearAllCmdModulePinzaCompleta(AspirazioneDX1,AspirazioneSX1,AspirazioneDX2,AspirazioneSX2,CilindroApertura,CilindroSbloccoRotazione,CilindroSbloccoBascolante,AspirazioneFaldaDX,AspirazioneFaldaSX);			TFError(ErrCMDTIMEOUT,ErrNULL,ADR(CmdExe),ADR(State),ADR(Error),ADR(ErrorLog));
		END_IF


	ELSE
		TFError(ErrNOCMD,ErrNULL,ADR(CmdExe),ADR(State),ADR(Error),ADR(ErrorLog));

END_CASE;


(* ******************************************************************************************************** *)
(* State Input/Output *)
(* ******************************************************************************************************** *)
(* Fill Input/Output bit with sensor, electrovalve, etc. status *)

StatoPinza.LatoDxAperto 			:= CilindroApertura^.Status.Active;
StatoPinza.LatoDxChiuso 			:= CilindroApertura^.Status.Inactive;
StatoPinza.LatoSxAperto				:= CilindroApertura^.Status.Active;
StatoPinza.LatoSxChiuso				:= CilindroApertura^.Status.Inactive;

StatoPinza.LatoDxFaldaInPresa		:= AspirazioneFaldaDX^.Status.Active AND IN.TastoreCartoneDX AND NOT AspirazioneDX1^.Status.DepressioneSoglia1_OK AND NOT AspirazioneDX2^.Status.DepressioneSoglia1_OK AND FTC_FaldaDXFiltrata;
StatoPinza.LatoDxPiastrellaInPresa	:= (AspirazioneDX1^.Status.DepressioneSoglia1_OK AND AspirazioneDX2^.Status.DepressioneSoglia1_OK)  OR (IN.ByPassSensoreVuoto AND StatoPinza.ElementoPrelevato);// AND NOT IN.TastoreCartoneDX;
StatoPinza.LatoSxFaldaInPresa		:= AspirazioneFaldaSX^.Status.Active AND IN.TastoreCartoneSX AND NOT AspirazioneSX1^.Status.DepressioneSoglia1_OK AND NOT AspirazioneSX2^.Status.DepressioneSoglia1_OK AND FTC_FaldaSXFiltrata;
StatoPinza.LatoSxPiastrellaInPresa	:=(AspirazioneSX1^.Status.DepressioneSoglia1_OK AND AspirazioneSX2^.Status.DepressioneSoglia1_OK)  OR (IN.ByPassSensoreVuoto AND StatoPinza.ElementoPrelevato);// AND  IN.TastoreCartoneSX;
StatoPinza.RotazioneBloccata		:= CilindroSbloccoRotazione^.Status.Inactive;
StatoPinza.RotazioneSbloccata 		:= CilindroSbloccoRotazione^.Status.Active;

StatoPinza.LetturaFTC0 := DistanzaFTC0;
StatoPinza.LetturaFTC180 := DistanzaFTC180;
StatoPinza.LetturaFTC0_2 := DistanzaFTC0_2;
StatoPinza.LetturaFTC180_2 := DistanzaFTC180_2;

(* ******************************************************************************************************** *)
(* Input *)
(* ******************************************************************************************************** *)

(* ******************************************************************************************************** *)
(* Alarm *)
(* ******************************************************************************************************** *)

(* ******************************************************************************************************** *)
(* Error Check - Clear All Output!!! *)
(* ******************************************************************************************************** *)
IF Error.Code > ErrNULL THEN
	IF CmdExe.Code <> CmdNOP THEN
		IF CmdExe.Code <> CmdSTOP AND
			CmdExe.Code <> CmdPOWER AND
			CmdExe.Code <> CmdRESET AND
			CmdExe.Code <> CmdMAN AND
			CmdExe.Code <> CmdLOAD AND
			CmdExe.Code <> CmdUNLOAD THEN
			TFCommandClear(ADR(CmdNext));
			TFCommandExeClear(ADR(CmdExe));

			(* Clear All Output Here *)

		END_IF;
	END_IF;
END_IF;


(* ******************************************************************************************************** *)
(* Common Outputs *)
(* ******************************************************************************************************** *)

END_FUNCTION_BLOCK

// ---- POUs/TFModules/Utility/TFClearAllCmdModulePinzaCompleta.TcPOU
FUNCTION TFClearAllCmdModulePinzaCompleta : bool
VAR_INPUT
	AspirazioneDX : POINTER TO TF_VacumOVEM;
	AspirazioneSX : POINTER TO TF_VacumOVEM;
	AspirazioneDX2 : POINTER TO TF_VacumOVEM;
	AspirazioneSX2 : POINTER TO TF_VacumOVEM;

	CilindroApertura 			: POINTER TO DC_Cylinder;
	CilindroSbloccoRotazione 	: POINTER TO SC_Cylinder;
	CilindroSbloccoBascolante 	: POINTER TO SC_Cylinder;
	AspirazioneFaldaDX 			: POINTER TO SC_Cylinder;
	AspirazioneFaldaSX 			: POINTER TO SC_Cylinder;
END_VAR
VAR
END_VAR

TFOVEMClearAllCommand(AspirazioneDX^.Command);
TFOVEMClearAllCommand(AspirazioneSX^.Command);
TFOVEMClearAllCommand(AspirazioneDX2^.Command);
TFOVEMClearAllCommand(AspirazioneSX2^.Command);
TFCylinder_ClearAllCommand(ADR(CilindroApertura^.Command));
TFCylinder_ClearAllCommand(ADR(CilindroSbloccoRotazione^.Command));
TFCylinder_ClearAllCommand(ADR(AspirazioneFaldaDX^.Command));
TFCylinder_ClearAllCommand(ADR(AspirazioneFaldaSX^.Command));
TFCylinder_ClearAllCommand(ADR(CilindroSbloccoBascolante^.Command));

END_FUNCTION

// ---- POUs/TFModules/Utility/TFOVEMClearAllCommand.TcPOU
FUNCTION TFOVEMClearAllCommand : bool
VAR_INPUT
Command : POINTER TO Ovem_Command;
END_VAR
VAR
END_VAR

Command^.ErrorReset := FALSE;
Command^.Aspirazione_OFF:=FALSE;
Command^.Aspirazione_ON :=FALSE;
Command^.Aspirazione_ON_ScritturaSoglia:=FALSE;
Command^.ErrorReset := FALSE;
Command^.ErrorReset := FALSE;
Command^.ScriviParametri:= FALSE;

TFOVEMClearAllCommand:=TRUE;

END_FUNCTION

// ---- POUs/TFModules/Utility/TFCylinder_ClearAllCommand.TcPOU
FUNCTION TFCylinder_ClearAllCommand : bool
VAR_INPUT
Command : pointer to  CylinderCommand;
END_VAR
VAR
END_VAR

Command^.ErrorReset := FALSE;
Command^.Deactivation:=FALSE;
Command^.Activation:=FALSE;
Command^.Hold:=FALSE;
Command^.Abort:=FALSE;
Command^.Stop:= FALSE;
TFCylinder_ClearAllCommand:=TRUE;

END_FUNCTION

// ---- POUs/TFPalletizerData_Lastre/TFWAM_CreaMissione_DepPrelElemento.TcPOU
(* FB per il calcolo delle quote di deposito di un elemento *)
FUNCTION_BLOCK TFWAM_CreaMissione_DepPrelElemento
VAR_INPUT

	NPosInLavoro	: UINT; //Numero Postazione di depositio
	Angolo_Destinazione : LREAL; //Angolo di destinazione dell'elemento
	
	PosizioneAttuale_X : LREAL; //Posizione attuale asse X
	
	TipologiaTraiettoria : e_Tipo_Traiettoria; //Tipologia Traiettoria: con o senza approccio
	
	CicloDiPRelievo : BOOL;//Indica se la tipologia di ciclo è un prelievo
		
	Apprendimento : TFMachinePalletizer_CoordinateApprendimento;
	
	Offset_Apprendimento_X : REAL; //Offset X Apprendimento
	Offset_Apprendimento_Y : REAL; //Offset Y Apprendimento
	Offset_Apprendimento_Z : REAL; //Offset Z Apprendimento
	Offset_Apprendimento_J : REAL; //Offset J Apprendimento
	
	Quota_PostX		: LREAL; //Quota X Postazione
	Quota_PostY		: LREAL; //Quota Y Postazione
	Quota_PostZ		: LREAL; //Quota Z Postazione
	Quota_PostJ		: LREAL; //Quota J Postazione
	
	Offset_Postazione_X : REAL; //Offset X Postazione
	Offset_Postazione_Y : REAL; //Offset Y Postazione
	Offset_Postazione_Z : REAL; //Offset Z Postazione
	Offset_Postazione_J : REAL; //Offset J Postazione
	
	Pallet_DimX				: LREAL; //Dimensione X Pallet
	Pallet_DimY				: LREAL; //Dimensione Y Pallet
	Pallet_DimZ				: LREAL; //Dimensione Z Pallet
	Pallet_DimBaseUtile		: LREAL; //Dimensione Y Base Util

	HmaxElemento	: LREAL;//Indica l'altezza massima dell'elemento,serve per i cicli di prelievo in cassa e pallet per determiinare le quote di approccio

	
	Offset_Pallet_X_0		: LREAL; //Offset X Pallet o Casse
	Offset_Pallet_Y_0		: LREAL; //Offset Y Pallet o Casse 
	Offset_Pallet_Z_0		: LREAL; //Offset Z Pallet o Casse + è grande + il deposito si distanzia dal supporto
	Offset_Pallet_J_0		: LREAL; //Offset J Pallet o Casse + è grande + la lastra sarà inclinata verso l'angolo crescente
	
	Offset_Pallet_X_90		: LREAL; //Offset X Pallet lato 0-90 
	Offset_Pallet_Y_90		: LREAL; //Offset Y Pallet lato 0-90 + è grande + il deposito si distanzia dal supporto
	Offset_Pallet_Z_90		: LREAL; //Offset Z Pallet lato 0-90 + è grande + il deposito si distanzia dal supporto
	Offset_Pallet_J_90		: LREAL; //Offset J Pallet lato 0-90 + è grande + la lastra sarà inclinata in fase di deposito
	
	Offset_Pallet_X_180		: LREAL; //Offset X Pallet lato 90-180
	Offset_Pallet_Y_180		: LREAL; //Offset Y Pallet lato 90-180 + è grande + il deposito si distanzia dal supporto
	Offset_Pallet_Z_180		: LREAL; //Offset Z Pallet lato 90-180 + è grande + il deposito si distanzia dal supporto
	Offset_Pallet_J_180		: LREAL; //Offset J Pallet lato 90-180 + è grande + la lastra sarà inclinata in fase di deposito
	
	Quota_FormaturaX 		: LREAL; //Quota Deposito X da Formatura
	Quota_FormaturaY 		: LREAL; //Quota Deposito Y da Formatura
	Quota_FormaturaZ 		: LREAL; //Quota Deposito Z da Formatura
	Quota_FormaturaJ 		: LREAL; //Quota Deposito Z da Formatura
	
	Distanza_ApproccioFormaturaX 		: LREAL; //Approccio in direzione X
	Distanza_ApproccioFormaturaY 		: LREAL; //Approccio in direzione Y
	Distanza_ApproccioFormaturaZ 		: LREAL; //Approccio in direzione Z
	Distanza_ApproccioFormaturaJ 		: LREAL; //Approccio in direzione J
	
END_VAR
VAR_OUTPUT
	
	Quota_DestX : LREAL; // Quota DESTINAZIONE X
	Quota_DestY : LREAL; // Quota DESTINAZIONE Y
	Quota_DestZ : LREAL; // Quota DESTINAZIONE Z
	Quota_DestJ : LREAL; // Quota DESTINAZIONE J
	
	Quota_ApproccioDestX : LREAL; // Quota Approccio DESTINAZIONE X
	Quota_ApproccioDestY : LREAL; // Quota Approccio DESTINAZIONE Y
	Quota_ApproccioDestZ : LREAL; // Quota Approccio DESTINAZIONE Z
	Quota_ApproccioDestJ : LREAL; // Quota Approccio DESTINAZIONE J
	
	Errore : TFError_WAM;
END_VAR
VAR
	Quota_DestYEnFun0: REAL;
	Quota_DestYEnFun180: REAL;
END_VAR

Errore.Code := 0;

CASE VERSO_PALLETTIZZATORE OF
	
	

	{region " Pallettizzatore DX "}					
	PALLETTIZZATORE_DX:
		CASE RIFERIMENTO_POSTAZIONE_WA OF
			{Region "ANGOLO DX" }
			ANGOLO_DX:
			
				(*******************************************************************************************************************)
(* Deposito su LASTRA con rotazione piano >90° e < 180°*)
				(*******************************************************************************************************************)																		
				IF Angolo_Destinazione > 90 THEN
					
					Quota_DestX	:= Quota_PostX + 						(* Quota X Postazione *)
									Offset_Postazione_X + 				(* Offset Postazione *)
									//Pallet_DimX/2 +						(* Dimensione/2 del Pallet/Cassa/Cavallina *)
									Offset_Pallet_X_180 +				(* Offset Deposito Direzione X del pallet *)
									Quota_FormaturaX;					(* Quota di deposito X da Formatura *)
				
					Quota_DestY := Quota_PostY + 						(* Quota Y Postazione *)
									IngombroDestinazioneY_Neg +
									Offset_Postazione_Y + 				(* Offset Postazione *)																								
									//Pallet_DimY/2 -						(* Dimensione/2 del Pallet/Cassa/Cavallina *)
									Offset_Pallet_Y_180 +				(* Offset Deposito Direzione Y del pallet *)
									Quota_FormaturaY; 					(* Quota di deposito Y da Formatura *)
										
					Quota_DestZ	:= Quota_PostZ + 						(* Quota Y Postazione *)
									Offset_Postazione_Z +				(* Offset Postazione *)	
									//Pallet_DimZ +						(* Dimensione/2 del Pallet/Cassa/Cavallina *)
									Offset_Pallet_Z_180 + 				(* Offset Deposito Direzione Z del pallet *)
									(-ScostamentoVerticalePuntoCentrale)+(* Sporgenza rispetto al filo pinza quando è in orizzontale *)
									Quota_FormaturaZ;					(* Quota di deposito Z da Formatura *)
							
					Quota_DestJ	:= Quota_FormaturaJ +					(* Quota di deposito Z da Formatura *)
									Offset_Pallet_J_180;				(* Offset Deposito inclinazione J del pallet *)
					
					(* Se ho l'abilitazione dell'utilizzo delle quote apprese,
						LE utilizzo come quote "buone" per eseguire il posizionamento *)				
					//Posizionamento lungo X
					IF Apprendimento.X.Lato180.Stato = APPRENDIMENTO_ESEGUITO THEN
						Quota_DestX := Apprendimento.X.Lato180.QuotaRilevata;
					END_IF
					//Posizionamento lungo Y lato 180°
					IF Apprendimento.Y.Lato180.Stato = APPRENDIMENTO_ESEGUITO THEN
						Quota_DestY := Apprendimento.Y.Lato180.QuotaRilevata;
					END_IF
					//Posizionamento lungo Z
					IF Apprendimento.Z.Lato180.Stato = APPRENDIMENTO_ESEGUITO THEN
						Quota_DestZ := Apprendimento.Z.Lato180.QuotaRilevata;
					END_IF
					//Posizionamento lungo J lato 180°
					IF Apprendimento.J.Lato180.Stato = APPRENDIMENTO_ESEGUITO THEN
						Quota_DestJ := Apprendimento.J.Lato180.QuotaRilevata;
					END_IF			
				(*****************************************************************************************************************)
				(************************************************ QUOTE APPROCCIO ************************************************)
				(*****************************************************************************************************************)	
					
					(* Valutazione della Direzione dell'Asse X*)
					IF PosizioneAttuale_X >= Quota_DestX THEN // La posizione attuale è maggiore della posizione di destinazione 
						Quota_ApproccioDestX := Quota_DestX +					(* Quota di deposito X *)
												Distanza_ApproccioFormaturaX;		(* Approccio X da Formatura *)	
					ELSE // La posizione attuale è minore della posizione di destinazione 
						Quota_ApproccioDestX := Quota_DestX -					(* Quota di deposito X *)
												Distanza_ApproccioFormaturaX;		(* Approccio X da Formatura *)
					END_IF			
				
					Quota_ApproccioDestY := Quota_DestY + 						(* Quota di deposito Y *)
											Distanza_ApproccioFormaturaY; 			(* Approccio Y da Formatura *)
										
					Quota_ApproccioDestZ := Quota_DestZ +						(* Quota di deposito Z da Formatura *)
											Distanza_ApproccioFormaturaZ;			(* Approccio Z da Formatura *)
							
					Quota_ApproccioDestJ := Quota_DestJ +						(* Quota di deposito J da Formatura *)
											Distanza_ApproccioFormaturaJ;			(* Approccio J da Formatura *)
									
				(*******************************************************************************************************************)						
											(* Deposito su LASTRA con rotazione piano < 90° e >0°*)	
				(*******************************************************************************************************************)							
				ELSIF Angolo_Destinazione < 90 THEN
					
					Quota_DestX	:= Quota_PostX + 						(* Quota X Postazione *)
									Offset_Postazione_X + 				(* Offset Postazione *)
									//Pallet_DimX/2 +						(* Dimensione/2 del Pallet/Cassa/Cavallina *)
									Offset_Pallet_X_0 +					(* Offset Deposito Direzione X del pallet *)
									Quota_FormaturaX;					(* Quota di deposito X da Formatura *)
				
					Quota_DestY := Quota_PostY - 						(* Quota Y Postazione *)
									IngombroDestinazioneY_Pos +
									Offset_Postazione_Y - 				(* Offset Postazione *)																							
									Pallet_DimY/2 -						(* Dimensione/2 del Pallet/Cassa/Cavallina *)
									Offset_Pallet_Y_0 +					(* Offset Deposito Direzione Y del pallet *)
									Quota_FormaturaY; 					(* Quota di deposito Y da Formatura *)
										
					Quota_DestZ	:= Quota_PostZ + 						(* Quota Y Postazione *)
									Offset_Postazione_Z +				(* Offset Postazione *)	
									//Pallet_DimZ +
									Offset_Pallet_Z_0 + 				(* Offset Deposito Direzione Z del pallet *)
									(-ScostamentoVerticalePuntoCentrale) +		(* Sporgenza rispetto al filo pinza quando è in orizzontale *)
									Quota_FormaturaZ;					(* Quota di deposito Z da Formatura *)
							
					Quota_DestJ	:= Quota_FormaturaJ +					(* Quota di deposito Z da Formatura *)
									Offset_Pallet_J_0;					(* Offset Deposito inclinazione J del pallet *)
					
					Apprendimento.Y.Lato0.Stato := APPRENDIMENTO_DA_ESEGUIRE ;		  
										
												  
															
					(* Se ho l'abilitazione dell'utilizzo delle quote apprese,
						LE utilizzo come quote "buone" per eseguire il posizionamento *)				
					//Posizionamento lungo X
					IF Apprendimento.X.Lato0.Stato = APPRENDIMENTO_ESEGUITO THEN
						Quota_DestX := Apprendimento.X.Lato0.QuotaRilevata;
					END_IF
					//Posizionamento lungo Y lato 0°
					IF Apprendimento.Y.Lato0.Stato = APPRENDIMENTO_ESEGUITO THEN
						Quota_DestY := Apprendimento.Y.Lato0.QuotaRilevata;
					END_IF
					//Posizionamento lungo Z
					IF Apprendimento.Z.Lato0.Stato = APPRENDIMENTO_ESEGUITO THEN
						Quota_DestZ := Apprendimento.Z.Lato0.QuotaRilevata;
					END_IF
					//Posizionamento lungo J lato 0°
					IF Apprendimento.J.Lato0.Stato = APPRENDIMENTO_ESEGUITO THEN
						Quota_DestJ := Apprendimento.J.Lato0.QuotaRilevata;
					END_IF		
				(*****************************************************************************************************************)
				(************************************************ QUOTE APPROCCIO ************************************************)
				(*****************************************************************************************************************)	
					
					(* Valutazione della Direzione dell'Asse X*)
					IF PosizioneAttuale_X >= Quota_DestX THEN // La posizione attuale è maggiore della posizione di destinazione 
						Quota_ApproccioDestX := Quota_DestX +					(* Quota di deposito X *)
												Distanza_ApproccioFormaturaX;		(* Approccio X da Formatura *)	
					ELSE // La posizione attuale è minore della posizione di destinazione 
						Quota_ApproccioDestX := Quota_DestX -					(* Quota di deposito X *)
												Distanza_ApproccioFormaturaX;		(* Approccio X da Formatura *)
					END_IF			
				
					Quota_ApproccioDestY := Quota_DestY - 						(* Quota di deposito Y *)
											Distanza_ApproccioFormaturaY; 			(* Approccio Y da Formatura *)
										
					Quota_ApproccioDestZ := Quota_DestZ +						(* Quota di deposito Z *)
											Distanza_ApproccioFormaturaZ;			(* Approccio Z da Formatura *)
							
					Quota_ApproccioDestJ := Quota_DestJ +						(* Quota di deposito J *)
											Distanza_ApproccioFormaturaJ;			(* Approccio J da Formatura *)				
							
				(*******************************************************************************************************************)						
											(* Deposito su LASTRA in cassa con rotazione piano = 90° *)
				(*******************************************************************************************************************)
				ELSE
					
					Quota_DestX	:= Quota_PostX + 						(* Quota X Postazione *)
									Offset_Postazione_X + 				(* Offset Postazione *)
									Pallet_DimX/2 +						(* Dimensione/2 del Pallet/Cassa/Cavallina *)
									Offset_Pallet_X_90;// +				(* Offset Deposito Direzione X del pallet *)
									//;Quota_FormaturaX;					(* Quota di deposito X da Formatura *)
														
					Quota_DestY := Quota_PostY + 						(* Quota Y Postazione *)
									Offset_Postazione_Y + 				(* Offset Postazione *)																							
									Pallet_DimY/2 +						(* Dimensione/2 del Pallet/Cassa/Cavallina *)
									Offset_Pallet_Y_90;// +				(* Offset Deposito Direzione Y del pallet *)
									//Quota_FormaturaY; 					(* Quota di deposito Y da Formatura *)
											
					Quota_DestZ	:= Quota_PostZ + 						(* Quota Y Postazione *)
									Offset_Postazione_Z +				(* Offset Postazione *)	
									//Pallet_DimZ +						(* Dimensione/2 del Pallet/Cassa/Cavallina *)
									Offset_Pallet_Z_90 + 				(* Offset Deposito Direzione Z del pallet *)
									Quota_FormaturaZ;					(* Quota di deposito Z da Formatura *)										
					Quota_DestJ	:= Quota_FormaturaJ +					(* Quota di deposito Z da Formatura *)
									Offset_Pallet_J_90;					(* Offset Deposito inclinazione J del pallet *)
					
					(* Se ho l'abilitazione dell'utilizzo delle quote apprese,
						LE utilizzo come quote "buone" per eseguire il posizionamento *)				
				//Posizionamento lungo X
					IF Apprendimento.X.Lato90.Stato = APPRENDIMENTO_ESEGUITO THEN
						Quota_DestX := Apprendimento.X.Lato90.QuotaRilevata;
					END_IF
					//Posizionamento lungo Y lato 90°
					IF Apprendimento.Y.Lato90.Stato = APPRENDIMENTO_ESEGUITO THEN
						Quota_DestY := Apprendimento.Y.Lato90.QuotaRilevata;
					END_IF
					//Posizionamento lungo Z
					IF Apprendimento.Z.Lato90.Stato <> APPRENDIMENTO_DISABILITATO THEN
						IF Apprendimento.Z.Lato90.Stato = APPRENDIMENTO_ESEGUITO THEN
							Quota_ApproccioDestZ := Apprendimento.Z.Lato90.QuotaRilevata + Distanza_ApproccioFormaturaZ;
						ELSE
							Quota_ApproccioDestZ := Apprendimento.Z.Lato90.QuotaStart + Offset_Apprendimento_Z;
						END_IF
					ELSE
						Quota_ApproccioDestZ := Quota_DestZ +						(* Quota di deposito Z *)
												Distanza_ApproccioFormaturaZ;			(* Approccio Z da Formatura *)
					END_IF
					//Posizionamento lungo J lato 0°
					IF Apprendimento.J.Lato90.Stato = APPRENDIMENTO_ESEGUITO THEN
						Quota_DestJ := Apprendimento.J.Lato90.QuotaRilevata;
					END_IF		
				(*****************************************************************************************************************)
				(************************************************ QUOTE APPROCCIO ************************************************)
				(*****************************************************************************************************************)										
					Quota_ApproccioDestX	:= Quota_DestX;				(* Quota di deposito X *)
														
					Quota_ApproccioDestY 	:= Quota_DestY; 			(* Quota di deposito Y *)
											
					//Quota_ApproccioDestZ := Quota_DestZ +						(* Quota di deposito Z *)
					//						Distanza_ApproccioFormaturaZ;			(* Approccio Z da Formatura *)
										
					Quota_ApproccioDestJ	:= Quota_DestJ;				(* Quota di deposito J *)				
					
				END_IF
			{endregion}
			{Region "CENTRALE" }				
			CENTRALE :
				(*******************************************************************************************************************)
											(* Deposito su LASTRA con rotazione piano >90° e < 180°*)
				(*******************************************************************************************************************)																		
				IF Angolo_Destinazione > 90 THEN
					Quota_DestX	:= Quota_PostX + 						(* Quota X Postazione *)
									Offset_Postazione_X + 				(* Offset Postazione *)
									Offset_Pallet_X_180;// +				(* Offset Deposito Direzione X del pallet *)
									//Quota_FormaturaX;					(* Quota di deposito X da Formatura *)
				
					Quota_DestY := Quota_PostY + 						(* Quota Y Postazione *)
									IngombroDestinazioneY_Neg +
									Offset_Postazione_Y + 				(* Offset Postazione *)																							
									Offset_Pallet_Y_180 +				(* Offset Deposito Direzione Y del pallet !!!!!*)
									ABS(Quota_FormaturaY); 					(* Quota di deposito Y da Formatura !!!!!!!*)
										
					Quota_DestZ	:= Quota_PostZ + 						(* Quota Y Postazione *)
									Offset_Postazione_Z +				(* Offset Postazione *)	
									//Pallet_DimZ +						(* Dimensione/2 del Pallet/Cassa/Cavallina *)
									Offset_Pallet_Z_180 + 				(* Offset Deposito Direzione Z del pallet *)
									(-ScostamentoVerticalePuntoCentrale) +		(* Sporgenza rispetto al filo pinza quando è in orizzontale *)
									Quota_FormaturaZ;					(* Quota di deposito Z da Formatura *)
							
					Quota_DestJ	:= Quota_FormaturaJ +					(* Quota di deposito Z da Formatura *)
									Offset_Pallet_J_180;				(* Offset Deposito inclinazione J del pallet *)
							
					(* Se ho l'abilitazione dell'utilizzo delle quote apprese,
						LE utilizzo come quote "buone" per eseguire il posizionamento *)				
					//Posizionamento lungo X
					IF Apprendimento.X.Lato180.Stato = APPRENDIMENTO_ESEGUITO THEN
						Quota_DestX := Apprendimento.X.Lato180.QuotaRilevata;
					END_IF
					//Posizionamento lungo Y lato 180°
					//IF Apprendimento.Y.Lato180.Stato = APPRENDIMENTO_ESEGUITO THEN
					//	Quota_DestY := Apprendimento.Y.Lato180.QuotaRilevata;
					//END_IF
					//Posizionamento lungo Z
					IF Apprendimento.Z.Lato180.Stato = APPRENDIMENTO_ESEGUITO THEN
						Quota_DestZ := Apprendimento.Z.Lato180.QuotaRilevata;
					END_IF
					//Posizionamento lungo J lato 180°
					IF Apprendimento.J.Lato180.Stato = APPRENDIMENTO_ESEGUITO THEN
						Quota_DestJ := Apprendimento.J.Lato180.QuotaRilevata;
					END_IF	
				(*****************************************************************************************************************)
				(************************************************ QUOTE APPROCCIO ************************************************)
				(*****************************************************************************************************************)										
					Quota_ApproccioDestX	:= Quota_DestX;				(* Quota di deposito X *)
														
					//Quota_ApproccioDestY 	:= Quota_DestY; 			(* Quota di deposito Y *)
					IF Apprendimento.Y.Lato180.Stato <> APPRENDIMENTO_DISABILITATO THEN
						IF Apprendimento.Y.Lato180.Stato = APPRENDIMENTO_ESEGUITO THEN
							Quota_ApproccioDestY := Apprendimento.Y.Lato180.QuotaRilevata + Distanza_ApproccioFormaturaY;
						ELSE
							Apprendimento.Y.Lato180.QuotaStart := Quota_DestY + (Pallet_DimY/2) +Offset_Apprendimento_Y; 		  
							Quota_ApproccioDestY := Apprendimento.Y.Lato180.QuotaStart + Offset_Apprendimento_Y;
						END_IF
					ELSE
						Quota_ApproccioDestY := Quota_DestY +						(* Quota di deposito Y *)
												Distanza_ApproccioFormaturaY;		(* Approccio Y da Formatura *)
					END_IF
											
					Quota_ApproccioDestZ 	:= Quota_DestZ; 			(* Quota di deposito Z *)
										
					Quota_ApproccioDestJ	:= Quota_DestJ;				(* Quota di deposito J *)
									
				(*******************************************************************************************************************)						
											(* Deposito su LASTRA con rotazione piano < 90° e >0°*)	
				(*******************************************************************************************************************)							
				ELSIF Angolo_Destinazione < 90 THEN
					
					Quota_DestX	:= Quota_PostX + 						(* Quota X Postazione *)
									Offset_Postazione_X + 				(* Offset Postazione *)
									Offset_Pallet_X_0;// +					(* Offset Deposito Direzione X del pallet *)
									//Quota_FormaturaX;					(* Quota di deposito X da Formatura *)
				
					Quota_DestY := Quota_PostY + 						(* Quota Y Postazione *)
									(-IngombroDestinazioneY_Pos)+
									Offset_Postazione_Y - 				(* Offset Postazione *)																								
									Offset_Pallet_Y_0 -					(* Offset Deposito Direzione Y del pallet *)
									ABS(Quota_FormaturaY); 					(* Quota di deposito Y da Formatura *)
										
					Quota_DestZ	:= Quota_PostZ + 						(* Quota Y Postazione *)
									Offset_Postazione_Z +				(* Offset Postazione *)	
									//Pallet_DimZ +						(* Dimensione/2 del Pallet/Cassa/Cavallina *)
									Offset_Pallet_Z_0 + 				(* Offset Deposito Direzione Z del pallet *)
									(-ScostamentoVerticalePuntoCentrale) +		(* Sporgenza rispetto al filo pinza quando è in orizzontale *)
									Quota_FormaturaZ;					(* Quota di deposito Z da Formatura *)
							
					Quota_DestJ	:= Quota_FormaturaJ +					(* Quota di deposito Z da Formatura *)
									Offset_Pallet_J_0;					(* Offset Deposito inclinazione J del pallet *)
				
					(* Se ho l'abilitazione dell'utilizzo delle quote apprese,
						LE utilizzo come quote "buone" per eseguire il posizionamento *)				
					//Posizionamento lungo X
					IF Apprendimento.X.Lato0.Stato = APPRENDIMENTO_ESEGUITO THEN
						Quota_DestX := Apprendimento.X.Lato0.QuotaRilevata;
					END_IF
					//Posizionamento lungo Y lato 0°
					IF Apprendimento.Y.Lato0.Stato = APPRENDIMENTO_ESEGUITO THEN
						Quota_DestY := Apprendimento.Y.Lato0.QuotaRilevata;
					END_IF
					//Posizionamento lungo Z
					IF Apprendimento.Z.Lato0.Stato = APPRENDIMENTO_ESEGUITO THEN
						Quota_DestZ := Apprendimento.Z.Lato0.QuotaRilevata;
					END_IF
					//Posizionamento lungo J lato 0°
					IF Apprendimento.J.Lato0.Stato = APPRENDIMENTO_ESEGUITO THEN
						Quota_DestJ := Apprendimento.J.Lato0.QuotaRilevata;
					END_IF
				(*****************************************************************************************************************)
				(************************************************ QUOTE APPROCCIO ************************************************)
				(*****************************************************************************************************************)										
					Quota_ApproccioDestX	:= Quota_DestX;				(* Quota di deposito X *)
														
					Quota_ApproccioDestY 	:= Quota_DestY; 			(* Quota di deposito Y *)
											
					Quota_ApproccioDestZ 	:= Quota_DestZ; 			(* Quota di deposito Z *)
										
					Quota_ApproccioDestJ	:= Quota_DestJ;				(* Quota di deposito J *)			
				(*******************************************************************************************************************)						
											(* Deposito su LASTRA in cassa con rotazione piano = 90° *)
				(*******************************************************************************************************************)
				ELSE
					
					Quota_DestX	:= Quota_PostX + 						(* Quota X Postazione *)
									Offset_Postazione_X + 				(* Offset Postazione *)
									Offset_Pallet_X_90;// +				(* Offset Deposito Direzione X del pallet *)
									//Quota_FormaturaX;					(* Quota di deposito X da Formatura *)
														
					Quota_DestY := Quota_PostY + 						(* Quota Y Postazione *)
									Offset_Postazione_Y + 				(* Offset Postazione *)																							
									Offset_Pallet_Y_90;// +				(* Offset Deposito Direzione Y del pallet *)
									//Quota_FormaturaY; 					(* Quota di deposito Y da Formatura *)
											
					Quota_DestZ	:= Quota_PostZ + 						(* Quota Y Postazione *)
									Offset_Postazione_Z +				(* Offset Postazione *)	
									//Pallet_DimZ +						(* Dimensione/2 del Pallet/Cassa/Cavallina *)
									Offset_Pallet_Z_90 + 				(* Offset Deposito Direzione Z del pallet *)
									Quota_FormaturaZ;					(* Quota di deposito Z da Formatura *)
										
					Quota_DestJ	:= Quota_FormaturaJ +					(* Quota di deposito Z da Formatura *)
									Offset_Pallet_J_90;					(* Offset Deposito inclinazione J del pallet *)
				
					(* Se ho l'abilitazione dell'utilizzo delle quote apprese,
						LE utilizzo come quote "buone" per eseguire il posizionamento *)				
					//Posizionamento lungo X
					//IF Apprendimento.X.Lato90.Stato = APPRENDIMENTO_ESEGUITO THEN
					//	Quota_DestX := Apprendimento.X.Lato90.QuotaRilevata;
					//END_IF
					////Posizionamento lungo Y lato 90°
					//IF Apprendimento.Y.Lato90.Stato = APPRENDIMENTO_ESEGUITO THEN
					//	Quota_DestY := Apprendimento.Y.Lato90.QuotaRilevata;
					//END_IF
					//Posizionamento lungo Z
					//Posizionamento lungo Z
					IF Apprendimento.Z.Lato90.Stato <> APPRENDIMENTO_DISABILITATO THEN
						IF Apprendimento.Z.Lato90.Stato = APPRENDIMENTO_ESEGUITO THEN
							Quota_ApproccioDestZ := Apprendimento.Z.Lato90.QuotaRilevata + Distanza_ApproccioFormaturaZ;
						ELSE
							Quota_ApproccioDestZ := Apprendimento.Z.Lato90.QuotaStart + Offset_Apprendimento_Z;
						END_IF
					ELSE
						Quota_ApproccioDestZ := Quota_DestZ +						(* Quota di deposito Z *)
												Distanza_ApproccioFormaturaZ;			(* Approccio Z da Formatura *)
					END_IF
					//Posizionamento lungo J lato 90°
					//IF Apprendimento.J.Lato90.Stato = APPRENDIMENTO_ESEGUITO THEN
					//	Quota_DestJ := Apprendimento.J.Lato90.QuotaRilevata;
					//END_IF			
				(*****************************************************************************************************************)
				(************************************************ QUOTE APPROCCIO ************************************************)
				(*****************************************************************************************************************)										
					Quota_ApproccioDestX	:= Quota_DestX;				(* Quota di deposito X *)
														
					Quota_ApproccioDestY 	:= Quota_DestY; 			(* Quota di deposito Y *)
											
					//Quota_ApproccioDestZ := Quota_DestZ +						(* Quota di deposito Z *)
					//						Distanza_ApproccioFormaturaZ;			(* Approccio Z da Formatura *)
										
					Quota_ApproccioDestJ	:= Quota_DestJ;				(* Quota di deposito J *)				
					
				END_IF
			{endregion}
			{Region "ANGOLO SX" }
			ANGOLO_SX :
				(*******************************************************************************************************************)
											(* Deposito su LASTRA con rotazione piano >90° e < 180°*)
				(*******************************************************************************************************************)
				IF Angolo_Destinazione > 90 THEN
					
					Quota_DestX	:= Quota_PostX + 						(* Quota X Postazione *)
									Offset_Postazione_X + 				(* Offset Postazione *)
									//Pallet_DimX/2 +						(* Dimensione/2 del Pallet/Cassa/Cavallina *)
									Offset_Pallet_X_180 +				(* Offset Deposito Direzione X del pallet *)
									(-Quota_FormaturaX);					(* Quota di deposito X da Formatura *)
				
					Quota_DestY := Quota_PostY + 						(* Quota Y Postazione *)
									IngombroDestinazioneY_Pos +
									Offset_Postazione_Y + 				(* Offset Postazione *)																							
									Pallet_DimY/2 +						(* Dimensione/2 del Pallet/Cassa/Cavallina *)
									Offset_Pallet_Y_180 +				(* Offset Deposito Direzione Y del pallet *)
									Quota_FormaturaY; 					(* Quota di deposito Y da Formatura *)
										
					Quota_DestZ	:= Quota_PostZ + 						(* Quota Y Postazione *)
									Offset_Postazione_Z +				(* Offset Postazione *)	
									//Pallet_DimZ +						(* Dimensione/2 del Pallet/Cassa/Cavallina *)
									Offset_Pallet_Z_180 + 				(* Offset Deposito Direzione Z del pallet *)
									(-ScostamentoVerticalePuntoCentrale) +		(* Sporgenza rispetto al filo pinza quando è in orizzontale *)
									Quota_FormaturaZ;					(* Quota di deposito Z da Formatura *)
							
					Quota_DestJ	:= Quota_FormaturaJ +					(* Quota di deposito Z da Formatura *)
									Offset_Pallet_J_180;				(* Offset Deposito inclinazione J del pallet *)
									
					(* Se ho l'abilitazione dell'utilizzo delle quote apprese,
						LE utilizzo come quote "buone" per eseguire il posizionamento *)				
					//Posizionamento lungo X
					IF Apprendimento.X.Lato180.Stato = APPRENDIMENTO_ESEGUITO THEN
						Quota_DestX := Apprendimento.X.Lato180.QuotaRilevata;
					END_IF
					//Posizionamento lungo Y lato 180°
					IF Apprendimento.Y.Lato180.Stato = APPRENDIMENTO_ESEGUITO THEN
						Quota_DestY := Apprendimento.Y.Lato180.QuotaRilevata;
					END_IF
					//Posizionamento lungo Z
					IF Apprendimento.Z.Lato180.Stato = APPRENDIMENTO_ESEGUITO THEN
						Quota_DestZ := Apprendimento.Z.Lato180.QuotaRilevata;
					END_IF
					//Posizionamento lungo J lato 180°
					IF Apprendimento.J.Lato180.Stato = APPRENDIMENTO_ESEGUITO THEN
						Quota_DestJ := Apprendimento.J.Lato180.QuotaRilevata;
					END_IF
				(*****************************************************************************************************************)
				(************************************************ QUOTE APPROCCIO ************************************************)
				(*****************************************************************************************************************)	
					
					(* Valutazione della Direzione dell'Asse X*)
					IF PosizioneAttuale_X >= Quota_DestX THEN // La posizione attuale è maggiore della posizione di destinazione 
						Quota_ApproccioDestX := Quota_DestX +					(* Quota di deposito X *)
												Distanza_ApproccioFormaturaX;		(* Approccio X da Formatura *)	
					ELSE // La posizione attuale è minore della posizione di destinazione 
						Quota_ApproccioDestX := Quota_DestX -					(* Quota di deposito X *)
												Distanza_ApproccioFormaturaX;		(* Approccio X da Formatura *)
					END_IF			
				
					Quota_ApproccioDestY := Quota_DestY + 						(* Quota di deposito Y *)
											Distanza_ApproccioFormaturaY; 			(* Approccio Y da Formatura *)
										
					Quota_ApproccioDestZ := Quota_DestZ +						(* Quota di deposito Z da Formatura *)
											Distanza_ApproccioFormaturaZ;			(* Approccio Z da Formatura *)
							
					Quota_ApproccioDestJ := Quota_DestJ +						(* Quota di deposito J da Forma*)	
											Distanza_ApproccioFormaturaJ;			(* Approccio J da Formatura *)
				(*******************************************************************************************************************)						
											(* Deposito su LASTRA con rotazione piano < 90° e >0°*)	
				(*******************************************************************************************************************)							
				ELSIF Angolo_Destinazione < 90 THEN
					
					Quota_DestX	:= Quota_PostX + 						(* Quota X Postazione *)
									Offset_Postazione_X + 				(* Offset Postazione *)
									//Pallet_DimX/2 +						(* Dimensione/2 del Pallet/Cassa/Cavallina *)
									Offset_Pallet_X_0 +					(* Offset Deposito Direzione X del pallet *)
									(-Quota_FormaturaX);					(* Quota di deposito X da Formatura *)
				
					Quota_DestY := Quota_PostY - 						(* Quota Y Postazione *)
									IngombroDestinazioneY_Pos +
									Offset_Postazione_Y + 				(* Offset Postazione *)																								
									Pallet_DimY/2 +						(* Dimensione/2 del Pallet/Cassa/Cavallina *)
									Offset_Pallet_Y_0 -					(* Offset Deposito Direzione Y del pallet *)
									Quota_FormaturaY; 					(* Quota di deposito Y da Formatura *)
										
					Quota_DestZ	:= Quota_PostZ + 						(* Quota Y Postazione *)
									Offset_Postazione_Z +				(* Offset Postazione *)	
									//Pallet_DimZ +						(* Dimensione/2 del Pallet/Cassa/Cavallina *)
									Offset_Pallet_Z_0 + 				(* Offset Deposito Direzione Z del pallet *)
									(-ScostamentoVerticalePuntoCentrale) +		(* Sporgenza rispetto al filo pinza quando è in orizzontale *)
									Quota_FormaturaZ;					(* Quota di deposito Z da Formatura *)
							
					Quota_DestJ	:= Quota_FormaturaJ +					(* Quota di deposito Z da Formatura *)
									Offset_Pallet_J_0;					(* Offset Deposito inclinazione J del pallet *)
									
					(* Se ho l'abilitazione dell'utilizzo delle quote apprese,
						LE utilizzo come quote "buone" per eseguire il posizionamento *)				
					//Posizionamento lungo X
					IF Apprendimento.X.Lato0.Stato = APPRENDIMENTO_ESEGUITO THEN
						Quota_DestX := Apprendimento.X.Lato0.QuotaRilevata;
					END_IF
					//Posizionamento lungo Y lato 0°
					IF Apprendimento.Y.Lato0.Stato = APPRENDIMENTO_ESEGUITO THEN
						Quota_DestY := Apprendimento.Y.Lato0.QuotaRilevata;
					END_IF
					//Posizionamento lungo Z
					IF Apprendimento.Z.Lato0.Stato = APPRENDIMENTO_ESEGUITO THEN
						Quota_DestZ := Apprendimento.Z.Lato0.QuotaRilevata;
					END_IF
					//Posizionamento lungo J lato 0°
					IF Apprendimento.J.Lato0.Stato = APPRENDIMENTO_ESEGUITO THEN
						Quota_DestJ := Apprendimento.J.Lato0.QuotaRilevata;
					END_IF
				(*****************************************************************************************************************)
				(************************************************ QUOTE APPROCCIO ************************************************)
				(*****************************************************************************************************************)	
					
					(* Valutazione della Direzione dell'Asse X*)
					IF PosizioneAttuale_X >= Quota_DestX THEN // La posizione attuale è maggiore della posizione di destinazione 
						Quota_ApproccioDestX := Quota_DestX +					(* Quota di deposito X *)
												Distanza_ApproccioFormaturaX;		(* Approccio X da Formatura *)	
					ELSE // La posizione attuale è minore della posizione di destinazione 
						Quota_ApproccioDestX := Quota_DestX -					(* Quota di deposito X *)
												Distanza_ApproccioFormaturaX;		(* Approccio X da Formatura *)
					END_IF			
				
					Quota_ApproccioDestY := Quota_DestY - 						(* Quota di deposito Y *)
											Distanza_ApproccioFormaturaY; 			(* Approccio Y da Formatura *)
										
					Quota_ApproccioDestZ := Quota_DestZ +						(* Quota di deposito Z *)
											Distanza_ApproccioFormaturaZ;			(* Approccio Z da Formatura *)
							
					Quota_ApproccioDestJ := Quota_DestJ +						(* Quota di deposito J *)
											Distanza_ApproccioFormaturaJ;			(* Approccio J da Formatura *)
							
				(*******************************************************************************************************************)						
											(* Deposito su LASTRA in cassa con rotazione piano = 90° *)
				(*******************************************************************************************************************)
				ELSE
					
					Quota_DestX	:= Quota_PostX + 						(* Quota X Postazione *)
									Offset_Postazione_X - 				(* Offset Postazione *)
									Pallet_DimX/2 +						(* Dimensione/2 del Pallet/Cassa/Cavallina *)
									Offset_Pallet_X_90;// -				(* Offset Deposito Direzione X del pallet *)
									//Quota_FormaturaX;					(* Quota di deposito X da Formatura *)
										
					Quota_DestY := Quota_PostY + 						(* Quota Y Postazione *)
									Offset_Postazione_Y + 				(* Offset Postazione *)																							
									Pallet_DimY/2 +						(* Dimensione/2 del Pallet/Cassa/Cavallina *)
									Offset_Pallet_Y_90;// +				(* Offset Deposito Direzione Y del pallet *)
									//Quota_FormaturaY; 					(* Quota di deposito Y da Formatura *)
											
					Quota_DestZ	:= Quota_PostZ + 						(* Quota Y Postazione *)
									Offset_Postazione_Z +				(* Offset Postazione *)	
									//Pallet_DimZ +						(* Dimensione/2 del Pallet/Cassa/Cavallina *)
									Offset_Pallet_Z_90 + 				(* Offset Deposito Direzione Z del pallet *)
									Quota_FormaturaZ;					(* Quota di deposito Z da Formatura *)
										
					Quota_DestJ	:= Quota_FormaturaJ;// +					(* Quota di deposito Z da Formatura *)
									//Offset_Pallet_J_90;					(* Offset Deposito inclinazione J del pallet *)
									
					(* Se ho l'abilitazione dell'utilizzo delle quote apprese,
						LE utilizzo come quote "buone" per eseguire il posizionamento *)				
					//Posizionamento lungo X
					IF Apprendimento.X.Lato90.Stato = APPRENDIMENTO_ESEGUITO THEN
						Quota_DestX := Apprendimento.X.Lato90.QuotaRilevata;
					END_IF
					//Posizionamento lungo Y lato 90°
					IF Apprendimento.Y.Lato90.Stato = APPRENDIMENTO_ESEGUITO THEN
						Quota_DestY := Apprendimento.Y.Lato90.QuotaRilevata;
					END_IF
					//Posizionamento lungo Z
					//Posizionamento lungo Z
					IF Apprendimento.Z.Lato90.Stato <> APPRENDIMENTO_DISABILITATO THEN
						IF Apprendimento.Z.Lato90.Stato = APPRENDIMENTO_ESEGUITO THEN
							Quota_ApproccioDestZ := Apprendimento.Z.Lato90.QuotaRilevata + Distanza_ApproccioFormaturaZ;
						ELSE
							Quota_ApproccioDestZ := Apprendimento.Z.Lato90.QuotaStart + Offset_Apprendimento_Z;
						END_IF
					ELSE
						Quota_ApproccioDestZ := Quota_DestZ +						(* Quota di deposito Z *)
												Distanza_ApproccioFormaturaZ;			(* Approccio Z da Formatura *)
					END_IF
					//Posizionamento lungo J lato 90°
					IF Apprendimento.J.Lato90.Stato = APPRENDIMENTO_ESEGUITO THEN
						Quota_DestJ := Apprendimento.J.Lato90.QuotaRilevata;
					END_IF
							
				(*****************************************************************************************************************)
				(************************************************ QUOTE APPROCCIO ************************************************)
				(*****************************************************************************************************************)										
					Quota_ApproccioDestX	:= Quota_DestX;				(* Quota di deposito X *)
														
					Quota_ApproccioDestY 	:= Quota_DestY; 			(* Quota di deposito Y *)
											
					//Quota_ApproccioDestZ := Quota_DestZ +						(* Quota di deposito Z *)
					//						Distanza_ApproccioFormaturaZ;			(* Approccio Z da Formatura *)
										
					Quota_ApproccioDestJ	:= Quota_DestJ;				(* Quota di deposito J *)				
					
				END_IF
			{endregion}
	
		ELSE
			Errore.Code := ErrWAM_FTC_PostazioneNONDefinita;
		END_CASE	
	{endregion}	
	{region " Pallettizzatore SX "}	
	PALLETTIZZATORE_SX:
		CASE RIFERIMENTO_POSTAZIONE_WA OF
			{Region "ANGOLO DX" }
			ANGOLO_DX:
			
				(*******************************************************************************************************************)
											(* Deposito su LASTRA con rotazione piano >90° e < 180°*)
				(*******************************************************************************************************************)																		
				IF Angolo_Destinazione > 90 THEN
					
					Quota_DestX	:= Quota_PostX + 						(* Quota X Postazione *)
									Offset_Postazione_X + 				(* Offset Postazione *)
									//Pallet_DimX/2 +						(* Dimensione/2 del Pallet/Cassa/Cavallina *)
									Offset_Pallet_X_180 +				(* Offset Deposito Direzione X del pallet *)
									(-Quota_FormaturaX);					(* Quota di deposito X da Formatura *)
				
					Quota_DestY := Quota_PostY + 						(* Quota Y Postazione *)
									IngombroDestinazioneY_Neg +
									Offset_Postazione_Y + 				(* Offset Postazione *)																								
									//Pallet_DimY/2 -						(* Dimensione/2 del Pallet/Cassa/Cavallina *)
									Offset_Pallet_Y_180 +				(* Offset Deposito Direzione Y del pallet *)
									Quota_FormaturaY; 					(* Quota di deposito Y da Formatura *)
										
					Quota_DestZ	:= Quota_PostZ + 						(* Quota Y Postazione *)
									Offset_Postazione_Z +				(* Offset Postazione *)	
									//Pallet_DimZ +						(* Dimensione/2 del Pallet/Cassa/Cavallina *)
									Offset_Pallet_Z_180 + 				(* Offset Deposito Direzione Z del pallet *)
									(-ScostamentoVerticalePuntoCentrale)+(* Sporgenza rispetto al filo pinza quando è in orizzontale *)
									Quota_FormaturaZ;					(* Quota di deposito Z da Formatura *)
							
					Quota_DestJ	:= Quota_FormaturaJ +					(* Quota di deposito Z da Formatura *)
									Offset_Pallet_J_180;				(* Offset Deposito inclinazione J del pallet *)
					
					(* Se ho l'abilitazione dell'utilizzo delle quote apprese,
						LE utilizzo come quote "buone" per eseguire il posizionamento *)				
					//Posizionamento lungo X
					IF Apprendimento.X.Lato180.Stato = APPRENDIMENTO_ESEGUITO THEN
						Quota_DestX := Apprendimento.X.Lato180.QuotaRilevata;
					END_IF
					//Posizionamento lungo Y lato 180°
					IF Apprendimento.Y.Lato180.Stato = APPRENDIMENTO_ESEGUITO THEN
						Quota_DestY := Apprendimento.Y.Lato180.QuotaRilevata;
					END_IF
					//Posizionamento lungo Z
					IF Apprendimento.Z.Lato180.Stato = APPRENDIMENTO_ESEGUITO THEN
						Quota_DestZ := Apprendimento.Z.Lato180.QuotaRilevata;
					END_IF
					//Posizionamento lungo J lato 180°
					IF Apprendimento.J.Lato180.Stato = APPRENDIMENTO_ESEGUITO THEN
						Quota_DestJ := Apprendimento.J.Lato180.QuotaRilevata;
					END_IF			
				(*****************************************************************************************************************)
				(************************************************ QUOTE APPROCCIO ************************************************)
				(*****************************************************************************************************************)	
					
					(* Valutazione della Direzione dell'Asse X*)
					IF PosizioneAttuale_X >= Quota_DestX THEN // La posizione attuale è maggiore della posizione di destinazione 
						Quota_ApproccioDestX := Quota_DestX +					(* Quota di deposito X *)
												Distanza_ApproccioFormaturaX;		(* Approccio X da Formatura *)	
					ELSE // La posizione attuale è minore della posizione di destinazione 
						Quota_ApproccioDestX := Quota_DestX -					(* Quota di deposito X *)
												Distanza_ApproccioFormaturaX;		(* Approccio X da Formatura *)
					END_IF			
				
					Quota_ApproccioDestY := Quota_DestY + 						(* Quota di deposito Y *)
											Distanza_ApproccioFormaturaY; 			(* Approccio Y da Formatura *)
										
					Quota_ApproccioDestZ := Quota_DestZ +						(* Quota di deposito Z da Formatura *)
											Distanza_ApproccioFormaturaZ;			(* Approccio Z da Formatura *)
							
					Quota_ApproccioDestJ := Quota_DestJ +						(* Quota di deposito J da Formatura *)
											Distanza_ApproccioFormaturaJ;			(* Approccio J da Formatura *)
									
				(*******************************************************************************************************************)						
											(* Deposito su LASTRA con rotazione piano < 90° e >0°*)	
				(*******************************************************************************************************************)							
				ELSIF Angolo_Destinazione < 90 THEN
					
					Quota_DestX	:= Quota_PostX + 						(* Quota X Postazione *)
									Offset_Postazione_X + 				(* Offset Postazione *)
									//Pallet_DimX/2 +						(* Dimensione/2 del Pallet/Cassa/Cavallina *)
									Offset_Pallet_X_0 +					(* Offset Deposito Direzione X del pallet *)
									(-Quota_FormaturaX);					(* Quota di deposito X da Formatura *)
				
					Quota_DestY := Quota_PostY - 						(* Quota Y Postazione *)
									IngombroDestinazioneY_Pos +
									Offset_Postazione_Y - 				(* Offset Postazione *)																							
									Pallet_DimY/2 -						(* Dimensione/2 del Pallet/Cassa/Cavallina *)
									Offset_Pallet_Y_0 -					(* Offset Deposito Direzione Y del pallet *)
									Quota_FormaturaY; 					(* Quota di deposito Y da Formatura *)
										
					Quota_DestZ	:= Quota_PostZ + 						(* Quota Y Postazione *)
									Offset_Postazione_Z +				(* Offset Postazione *)	
									//Pallet_DimZ +
									Offset_Pallet_Z_0 + 				(* Offset Deposito Direzione Z del pallet *)
									(-ScostamentoVerticalePuntoCentrale) +		(* Sporgenza rispetto al filo pinza quando è in orizzontale *)
									Quota_FormaturaZ;					(* Quota di deposito Z da Formatura *)
							
					Quota_DestJ	:= Quota_FormaturaJ +					(* Quota di deposito Z da Formatura *)
									Offset_Pallet_J_0;					(* Offset Deposito inclinazione J del pallet *)
					
					(* Se ho l'abilitazione dell'utilizzo delle quote apprese,
						LE utilizzo come quote "buone" per eseguire il posizionamento *)				
					//Posizionamento lungo X
					IF Apprendimento.X.Lato0.Stato = APPRENDIMENTO_ESEGUITO THEN
						Quota_DestX := Apprendimento.X.Lato0.QuotaRilevata;
					END_IF
					//Posizionamento lungo Y lato 0°
					IF Apprendimento.Y.Lato0.Stato = APPRENDIMENTO_ESEGUITO THEN
						Quota_DestY := Apprendimento.Y.Lato0.QuotaRilevata;
					END_IF
					//Posizionamento lungo Z
					IF Apprendimento.Z.Lato0.Stato = APPRENDIMENTO_ESEGUITO THEN
						Quota_DestZ := Apprendimento.Z.Lato0.QuotaRilevata;
					END_IF
					//Posizionamento lungo J lato 0°
					IF Apprendimento.J.Lato0.Stato = APPRENDIMENTO_ESEGUITO THEN
						Quota_DestJ := Apprendimento.J.Lato0.QuotaRilevata;
					END_IF		
				(*****************************************************************************************************************)
				(************************************************ QUOTE APPROCCIO ************************************************)
				(*****************************************************************************************************************)	
					
					(* Valutazione della Direzione dell'Asse X*)
					IF PosizioneAttuale_X >= Quota_DestX THEN // La posizione attuale è maggiore della posizione di destinazione 
						Quota_ApproccioDestX := Quota_DestX +					(* Quota di deposito X *)
												Distanza_ApproccioFormaturaX;		(* Approccio X da Formatura *)	
					ELSE // La posizione attuale è minore della posizione di destinazione 
						Quota_ApproccioDestX := Quota_DestX -					(* Quota di deposito X *)
												Distanza_ApproccioFormaturaX;		(* Approccio X da Formatura *)
					END_IF			
				
					Quota_ApproccioDestY := Quota_DestY - 						(* Quota di deposito Y *)
											Distanza_ApproccioFormaturaY; 			(* Approccio Y da Formatura *)
										
					Quota_ApproccioDestZ := Quota_DestZ +						(* Quota di deposito Z *)
											Distanza_ApproccioFormaturaZ;			(* Approccio Z da Formatura *)
							
					Quota_ApproccioDestJ := Quota_DestJ +						(* Quota di deposito J *)
											Distanza_ApproccioFormaturaJ;			(* Approccio J da Formatura *)				
							
				(*******************************************************************************************************************)						
											(* Deposito su LASTRA in cassa con rotazione piano = 90° *)
				(*******************************************************************************************************************)
				ELSE
					
					Quota_DestX	:= Quota_PostX + 						(* Quota X Postazione *)
									Offset_Postazione_X - 				(* Offset Postazione *)
									Pallet_DimX/2 +						(* Dimensione/2 del Pallet/Cassa/Cavallina *)
									Offset_Pallet_X_90;// +				(* Offset Deposito Direzione X del pallet *)
									//Quota_FormaturaX;					(* Quota di deposito X da Formatura *)
														
					Quota_DestY := Quota_PostY + 						(* Quota Y Postazione *)
									Offset_Postazione_Y + 				(* Offset Postazione *)																							
									Pallet_DimY/2 +						(* Dimensione/2 del Pallet/Cassa/Cavallina *)
									Offset_Pallet_Y_90;// +				(* Offset Deposito Direzione Y del pallet *)
									//Quota_FormaturaY; 					(* Quota di deposito Y da Formatura *)
											
					Quota_DestZ	:= Quota_PostZ + 						(* Quota Y Postazione *)
									Offset_Postazione_Z +				(* Offset Postazione *)	
									//Pallet_DimZ +						(* Dimensione/2 del Pallet/Cassa/Cavallina *)
									Offset_Pallet_Z_90 + 				(* Offset Deposito Direzione Z del pallet *)
									Quota_FormaturaZ;					(* Quota di deposito Z da Formatura *)										
					Quota_DestJ	:= Quota_FormaturaJ +					(* Quota di deposito Z da Formatura *)
									Offset_Pallet_J_90;					(* Offset Deposito inclinazione J del pallet *)
					
					(* Se ho l'abilitazione dell'utilizzo delle quote apprese,
						LE utilizzo come quote "buone" per eseguire il posizionamento *)				
				//Posizionamento lungo X
					IF Apprendimento.X.Lato90.Stato = APPRENDIMENTO_ESEGUITO THEN
						Quota_DestX := Apprendimento.X.Lato90.QuotaRilevata;
					END_IF
					//Posizionamento lungo Y lato 90°
					IF Apprendimento.Y.Lato90.Stato = APPRENDIMENTO_ESEGUITO THEN
						Quota_DestY := Apprendimento.Y.Lato90.QuotaRilevata;
					END_IF
					//Posizionamento lungo Z
					IF Apprendimento.Z.Lato90.Stato <> APPRENDIMENTO_DISABILITATO THEN
						IF Apprendimento.Z.Lato90.Stato = APPRENDIMENTO_ESEGUITO THEN
							Quota_ApproccioDestZ := Apprendimento.Z.Lato90.QuotaRilevata + Distanza_ApproccioFormaturaZ;
						ELSE
							Quota_ApproccioDestZ := Apprendimento.Z.Lato90.QuotaStart + Offset_Apprendimento_Z;
						END_IF
					ELSE
						Quota_ApproccioDestZ := Quota_DestZ +						(* Quota di deposito Z *)
												Distanza_ApproccioFormaturaZ;			(* Approccio Z da Formatura *)
					END_IF
					//Posizionamento lungo J lato 0°
					IF Apprendimento.J.Lato90.Stato = APPRENDIMENTO_ESEGUITO THEN
						Quota_DestJ := Apprendimento.J.Lato90.QuotaRilevata;
					END_IF		
				(*****************************************************************************************************************)
				(************************************************ QUOTE APPROCCIO ************************************************)
				(*****************************************************************************************************************)										
					Quota_ApproccioDestX	:= Quota_DestX;				(* Quota di deposito X *)
														
					Quota_ApproccioDestY 	:= Quota_DestY; 			(* Quota di deposito Y *)
											
					//Quota_ApproccioDestZ := Quota_DestZ +						(* Quota di deposito Z *)
					//						Distanza_ApproccioFormaturaZ;			(* Approccio Z da Formatura *)
										
					Quota_ApproccioDestJ	:= Quota_DestJ;				(* Quota di deposito J *)				
					
				END_IF
			{endregion}
			{Region "CENTRALE" }				
			CENTRALE :
				(*******************************************************************************************************************)
											(* Deposito su LASTRA con rotazione piano >90° e < 180°*)
				(*******************************************************************************************************************)																		
				IF Angolo_Destinazione > 90 THEN
					
					Quota_DestX	:= Quota_PostX + 						(* Quota X Postazione *)
									Offset_Postazione_X + 				(* Offset Postazione *)
									Offset_Pallet_X_180;// +				(* Offset Deposito Direzione X del pallet *)
									//Quota_FormaturaX;					(* Quota di deposito X da Formatura *)
				
					Quota_DestY := Quota_PostY + 						(* Quota Y Postazione *)
					(*MAX (IngombroDestinazioneY_Neg ,Dimensioni_Pinza.Spessore) + *)
					Dimensioni_Pinza.Spessore +
									Offset_Postazione_Y + 				(* Offset Postazione *)																							
									Offset_Pallet_Y_180 +				(* Offset Deposito Direzione Y del pallet *)
									Quota_FormaturaY; 					(* Quota di deposito Y da Formatura *)
											  
					Quota_DestYEnFun180 :=	Quota_DestY ;

				
					Quota_DestZ	:= Quota_PostZ + 						(* Quota Y Postazione *)
									Offset_Postazione_Z +				(* Offset Postazione *)	
									//Pallet_DimZ +						(* Dimensione/2 del Pallet/Cassa/Cavallina *)
									Offset_Pallet_Z_180 + 				(* Offset Deposito Direzione Z del pallet *)
									(-ScostamentoVerticalePuntoCentrale) +		(* Sporgenza rispetto al filo pinza quando è in orizzontale *)
									Quota_FormaturaZ;					(* Quota di deposito Z da Formatura *)
							
					Quota_DestJ	:= Quota_FormaturaJ +					(* Quota di deposito Z da Formatura *)
									Offset_Pallet_J_180;				(* Offset Deposito inclinazione J del pallet *)
							
					(* Se ho l'abilitazione dell'utilizzo delle quote apprese,
						LE utilizzo come quote "buone" per eseguire il posizionamento *)				
					//Posizionamento lungo X
					IF Apprendimento.X.Lato180.Stato = APPRENDIMENTO_ESEGUITO THEN
						Quota_DestX := Apprendimento.X.Lato180.QuotaRilevata;
					END_IF
					//Posizionamento lungo Y lato 180°
					IF Apprendimento.Y.Lato180.Stato = APPRENDIMENTO_ESEGUITO AND Temp_Bool[20] THEN
						Quota_DestY := Apprendimento.Y.Lato180.QuotaRilevata - 20;
					END_IF
					//Posizionamento lungo Z
					IF Apprendimento.Z.Lato180.Stato = APPRENDIMENTO_ESEGUITO THEN
						Quota_DestZ := Apprendimento.Z.Lato180.QuotaRilevata;
					END_IF
					//Posizionamento lungo J lato 180°
					IF Apprendimento.J.Lato180.Stato = APPRENDIMENTO_ESEGUITO THEN
						Quota_DestJ := Apprendimento.J.Lato180.QuotaRilevata;
					END_IF	
				(*****************************************************************************************************************)
				(************************************************ QUOTE APPROCCIO ************************************************)
				(*****************************************************************************************************************)										
					Quota_ApproccioDestX	:= Quota_DestX;				(* Quota di deposito X *)
														
					Quota_ApproccioDestY 	:= Quota_DestY; 			(* Quota di deposito Y *)
											
					Quota_ApproccioDestZ 	:= Quota_DestZ; 			(* Quota di deposito Z *)
										
					Quota_ApproccioDestJ	:= Quota_DestJ;				(* Quota di deposito J *)
									
				(*******************************************************************************************************************)						
											(* Deposito su LASTRA con rotazione piano < 90° e >0°*)	
				(*******************************************************************************************************************)							
				ELSIF Angolo_Destinazione < 90 THEN
					
					Quota_DestX	:= Quota_PostX + 						(* Quota X Postazione *)
									Offset_Postazione_X + 				(* Offset Postazione *)
									Offset_Pallet_X_0;// +					(* Offset Deposito Direzione X del pallet *)
									//Quota_FormaturaX;					(* Quota di deposito X da Formatura *)
				
					Quota_DestY := Quota_PostY + 						(* Quota Y Postazione *)
						(-MAX(IngombroDestinazioneY_Pos ,Dimensioni_Pinza.Spessore)) +
									Offset_Postazione_Y - 				(* Offset Postazione *)																								
									Offset_Pallet_Y_0 -					(* Offset Deposito Direzione Y del pallet *)
									Quota_FormaturaY (*-
									((Pallet_DimY/2 )- Pallet_DimBaseUtile)*)	; 					(* Quota di deposito Y da Formatura *)
					Quota_DestYEnFun0 :=	Quota_DestY ;				
					Quota_DestZ	:= Quota_PostZ + 						(* Quota Y Postazione *)
									Offset_Postazione_Z +				(* Offset Postazione *)	
									//Pallet_DimZ +						(* Dimensione/2 del Pallet/Cassa/Cavallina *)
									Offset_Pallet_Z_0 + 				(* Offset Deposito Direzione Z del pallet *)
									(-ScostamentoVerticalePuntoCentrale) +		(* Sporgenza rispetto al filo pinza quando è in orizzontale *)
									Quota_FormaturaZ;					(* Quota di deposito Z da Formatura *)
							
					Quota_DestJ	:= Quota_FormaturaJ +					(* Quota di deposito Z da Formatura *)
									Offset_Pallet_J_0;					(* Offset Deposito inclinazione J del pallet *)
				
					(* Se ho l'abilitazione dell'utilizzo delle quote apprese,
						LE utilizzo come quote "buone" per eseguire il posizionamento *)				
					//Posizionamento lungo X
				
	  
					IF Apprendimento.X.Lato0.Stato = APPRENDIMENTO_ESEGUITO THEN
						Quota_DestX := Apprendimento.X.Lato0.QuotaRilevata;
					END_IF
					//Posizionamento lungo Y lato 0°
					IF Apprendimento.Y.Lato0.Stato = APPRENDIMENTO_ESEGUITO AND Temp_Bool[20] THEN
						Quota_DestY := Apprendimento.Y.Lato0.QuotaRilevata;
					 
								   
					END_IF
					//Posizionamento lungo Z
					IF Apprendimento.Z.Lato0.Stato = APPRENDIMENTO_ESEGUITO THEN
						Quota_DestZ := Apprendimento.Z.Lato0.QuotaRilevata;
					END_IF
					//Posizionamento lungo J lato 0°
					IF Apprendimento.J.Lato0.Stato = APPRENDIMENTO_ESEGUITO THEN
						Quota_DestJ := Apprendimento.J.Lato0.QuotaRilevata;
					END_IF
				(*****************************************************************************************************************)
				(************************************************ QUOTE APPROCCIO ************************************************)
				(*****************************************************************************************************************)										
					Quota_ApproccioDestX	:= Quota_DestX;				(* Quota di deposito X *)
					IF 	Apprendimento.Y.Lato0.Stato = APPRENDIMENTO_ESEGUITO THEN
						Quota_ApproccioDestY 	:= Quota_DestY; 			(* Quota di deposito Y *)
					ELSE	
						Quota_ApproccioDestY  	:= Quota_DestY (*-100*); 			(* Quota di deposito Y *)	  
					END_IF								
					
											
					Quota_ApproccioDestZ 	:= Quota_DestZ; 			(* Quota di deposito Z *)
										
					Quota_ApproccioDestJ	:= Quota_DestJ;				(* Quota di deposito J *)			
				(*******************************************************************************************************************)						
											(* Deposito su LASTRA in cassa con rotazione piano = 90° *)
				(*******************************************************************************************************************)
				ELSE
					
					Quota_DestX	:= Quota_PostX + 						(* Quota X Postazione *)
									Offset_Postazione_X + 				(* Offset Postazione *)
									Offset_Pallet_X_90;// +				(* Offset Deposito Direzione X del pallet *)
									//Quota_FormaturaX;					(* Quota di deposito X da Formatura *)
														
					Quota_DestY := Quota_PostY + 						(* Quota Y Postazione *)
									Offset_Postazione_Y + 				(* Offset Postazione *)																							
									Offset_Pallet_Y_90;// +				(* Offset Deposito Direzione Y del pallet *)
									//Quota_FormaturaY; 					(* Quota di deposito Y da Formatura *)
											
